		Slew2AbsAzEl:=CmdResponseType.CommandActivated;	
	ELSE 
		Slew2AbsAzEl:=CmdResponseType.ParameterOutOfRange;
	END_IF			   
END_IF
r_write_position_az_out:=Pos_Az; // Writeing setpoint positions to Cyclic out put to get P.Set outputs
r_write_position_el_out:=Pos_El;
CommandArbiter.Status.LastCmdResponse:=Slew2AbsAzEl;
END_METHOD

METHOD Slew2AbsSingleAx : UINT
VAR_INPUT
	SessionID: UINT;
	Axis: Uint;
	Position:LREAL;
	Speed:LREAL;
END_VAR

VAR
END_VAR
CASE CommandArbiter.Status.DscCmdAuthority OF                    // Check that correct user is issueing a command
	LMC: IF SessionID= CommandArbiter.Lmc_ID THEN
			Slew2AbsSingleAx:= CmdResponseType.CommandActivated;
     	 END_IF
			
	EGUI: IF SessionID= CommandArbiter.Egui_ID THEN
			Slew2AbsSingleAx:= CmdResponseType.CommandActivated;
    	  END_IF		
ELSE 
     Slew2AbsSingleAx:= CmdResponseType.NoCmdAuth;
     Command_Arbiter_error:=1;	
END_CASE

IF Slew2AbsSingleAx = CmdResponseType.CommandActivated THEN // Dish State to see if move is possible
	Command_Arbiter_error:=0;
	//IF  Management.ErrorStatus.errGeneral=0 AND Management.WarningStatus.waMngmnt =0 THEN   If the Dish has errors that prevent movement then it will not be in a state where it can be moved. 
		CASE Management.Status.DscState OF 
			 DscStateType.Locked:        Slew2AbsSingleAx:=CmdResponseType.DishLocked;
			 DscStateType.Locked_Stowed: Slew2AbsSingleAx:=CmdResponseType.DishLocked;
			 DscStateType.Standstill:    Slew2AbsSingleAx:=CmdResponseType.CommandActivated;
		     DscStateType.Standby:       Slew2AbsSingleAx:=CmdResponseType.CommandActivated;
			 DscStateType.Stowed:	IF Axis=2 THEN 
				Slew2AbsSingleAx:= CmdResponseType.CommandActivated;
			ELSE
		 	Slew2AbsSingleAx:=CmdResponseType.Stowed;
			END_IF
  
		ELSE
		     Slew2AbsSingleAx:=CmdResponseType.CommandRejected;
		     Command_Arbiter_error:=1;
		END_CASE								
	//ELSE
	//	Slew2AbsAx:=CmdResponseType.CommandAborted;
	//	Command_Arbiter_error:=1;
	//END_IF
END_IF
	
IF Slew2AbsSingleAx = CmdResponseType.CommandActivated THEN  // Move selected axis
	b_goto_rel:=FALSE;
	CASE Axis OF 
		AxisSelectType.Az:	
            IF (Position <= gc_r_pos_max_Az) AND (Position>= gc_r_pos_min_Az) AND (Speed <= gc_r_vel_max_Az*6) THEN
           		b_activate_Az:=1;
			    r_goto_Az := LREAL_TO_REAL(Position);
				 IF Speed > r_vel_max_Az THEN    // For power management
					 r_goto_v_Az:= r_vel_max_Az;
				 ELSE
				 	 r_goto_v_Az:= LREAL_TO_REAL(Speed/6); 
				 END_IF
				b_stop_Az:= FALSE;
				b_start_goto_Az:= TRUE;
				Slew2AbsSingleAx:=CmdResponseType.CommandActivated;
				r_write_position_az_out:=Position; // Writeing setpoint positions to Cyclic out put to get P.Set outputs
			ELSE 
				Slew2AbsSingleAx:=CmdResponseType.ParameterOutOfRange;
			END_IF			   
		AxisSelectType.El:
 			IF (Position <= gc_r_pos_max_El) AND (Position>= gc_r_pos_min_El) AND (Speed <= gc_r_vel_max_El*6
) THEN
            	b_activate_el:=1;
				r_goto_El := LREAL_TO_REAL(Position);
				
				 IF Speed > r_vel_max_El THEN    // For power management
					 r_goto_v_El:= r_vel_max_El;
				 ELSE
				 	 r_goto_v_El:= LREAL_TO_REAL(Speed/6); 
				 END_IF
				
				b_stop_El:= FALSE;
				b_start_goto_El:= TRUE;
				Slew2AbsSingleAx:=CmdResponseType.CommandActivated;
				r_write_position_el_out:=Position; // Writeing setpoint positions to Cyclic out put to get P.Set outputs
			ELSE 
				Slew2AbsSingleAx:=CmdResponseType.ParameterOutOfRange;
			END_IF 
					    
		AxisSelectType.FI: 
			IF (Position <= gc_r_pos_max_Fi) AND (Position >= gc_r_pos_min_Fi) AND (Speed<= gc_r_vel_max_Fi*6) THEN
                 b_activate_Fi:=1;
				 r_goto_Fi := LREAL_TO_REAL(Position);
				 IF Speed > r_vel_max_Fi THEN 
					 r_goto_v_Fi:= r_vel_max_Fi;
				 ELSE
				 	 r_goto_v_Fi:= LREAL_TO_REAL(Speed/6); 
				 END_IF
				 b_stop_Fi:= FALSE;
				 b_start_goto_Fi:= TRUE;
				 Slew2AbsSingleAx:=CmdResponseType.CommandActivated;
				 r_write_position_fi_out:=Position; // Writeing setpoint positions to Cyclic out put to get P.Set outputs
		    ELSE 
				 Slew2AbsSingleAx:=CmdResponseType.ParameterOutOfRange;
			END_IF              
 			     									
	ELSE
		Slew2AbsSingleAx:=CmdResponseType.ParameterOutOfRange;
	END_CASE
END_IF

CommandArbiter.Status.LastCmdResponse:=Slew2AbsSingleAx;
END_METHOD

METHOD Slew2RelAzEl : UINT
VAR_INPUT
	SessionID:UINT;
	Pos_Az:LREAL;
	Pos_El:LREAL;
	Speed_Az:LREAL;
	Speed_El:LREAL;
	
END_VAR
CASE CommandArbiter.Status.DscCmdAuthority OF                    // Check that correct user is issueing a command
	LMC: IF SessionID= CommandArbiter.Lmc_ID THEN
			Slew2RelAzEl:= CmdResponseType.CommandActivated;
     	 END_IF
			
	EGUI: IF SessionID= CommandArbiter.Egui_ID THEN
			Slew2RelAzEl:= CmdResponseType.CommandActivated;
    	  END_IF		
ELSE 
     Slew2RelAzEl:= CmdResponseType.NoCmdAuth;
     Command_Arbiter_error:=1;	
END_CASE

IF Slew2RelAzEl = CmdResponseType.CommandActivated THEN // Dish State to see if move is possible
	Command_Arbiter_error:=0;
	//IF  Management.ErrorStatus.errGeneral=0 AND Management.WarningStatus.waMngmnt =0 THEN  (*The Dish in the standby state*)
		CASE Management.Status.DscState OF 
			 DscStateType.Locked:        Slew2RelAzEl:=CmdResponseType.DishLocked;
			 DscStateType.Locked_Stowed: Slew2RelAzEl:=CmdResponseType.DishLocked;
			 DscStateType.Standstill:    Slew2RelAzEl:=CmdResponseType.CommandActivated;
		     DscStateType.Standby:       Slew2RelAzEl:=CmdResponseType.CommandActivated;
			 DscStateType.Stowed:	     Slew2RelAzEl:=CmdResponseType.Stowed;
		ELSE
		     Slew2RelAzEl:=CmdResponseType.CommandRejected;
		     Command_Arbiter_error:=1;
		END_CASE								
	(*ELSE
		Slew2RelAzEl:=CmdResponseType.CommandAborted;
		Command_Arbiter_error:=1;
	END_IF *)
END_IF
	
IF Slew2RelAzEl = CmdResponseType.CommandActivated THEN  // Move selected axis
	IF (((Pos_Az + r_pos_az_v) <= gc_r_pos_max_Az) AND ((Pos_Az + r_pos_az_v )>= gc_r_pos_min_Az) AND ( Speed_Az <= gc_r_vel_max_Az*6)) AND (((Pos_El + r_pos_el_v) <= gc_r_pos_max_El) AND ((Pos_El + r_pos_el_v )>= gc_r_pos_min_El) AND ( Speed_El <= gc_r_vel_max_El*6)) THEN
    	b_activate_Az:=1;
		r_goto_Az := LREAL_TO_REAL(Pos_Az);
		b_goto_rel:=TRUE;
		r_goto_v_Az:= LREAL_TO_REAL(Speed_Az/6); 
		b_stop_Az:= FALSE;
		b_start_goto_Az:= TRUE;
		b_activate_el:=1;
		r_goto_El := LREAL_TO_REAL(Pos_El);
		r_goto_v_El:= LREAL_TO_REAL(Speed_El/6); 
		b_stop_El:= FALSE;
		b_start_goto_El:= TRUE;
		Slew2RelAzEl:=CmdResponseType.CommandActivated;	
	ELSE 
		Slew2RelAzEl:=CmdResponseType.ParameterOutOfRange;
	END_IF			   
	
END_IF

CommandArbiter.Status.LastCmdResponse:=Slew2RelAzEl;
END_METHOD

METHOD Slew2RelSingleAx : UINT
VAR_INPUT
	SessionID:UINT;
	Axis: UINT;
	Position:LREAL;
	Speed:LREAL;
END_VAR
CASE CommandArbiter.Status.DscCmdAuthority OF                    // Check that correct user is issueing a command
	LMC: IF SessionID= CommandArbiter.Lmc_ID THEN
			Slew2RelSingleAx:= CmdResponseType.CommandActivated;
     	 END_IF
			
	EGUI: IF SessionID= CommandArbiter.Egui_ID THEN
			Slew2RelSingleAx:= CmdResponseType.CommandActivated;
    	  END_IF		
ELSE 
     Slew2RelSingleAx:= CmdResponseType.NoCmdAuth;
     Command_Arbiter_error:=1;	
END_CASE

IF Slew2RelSingleAx = CmdResponseType.CommandActivated THEN // Dish State to see if move is possible
	Command_Arbiter_error:=0;
	//IF  Management.ErrorStatus.errGeneral=0 AND Management.WarningStatus.waMngmnt =0 THEN  (*The Dish in the standby state*)
		CASE Management.Status.DscState OF 
			 DscStateType.Locked:        Slew2RelSingleAx:=CmdResponseType.DishLocked;
			 DscStateType.Locked_Stowed: Slew2RelSingleAx:=CmdResponseType.DishLocked;
			 DscStateType.Standstill:    Slew2RelSingleAx:=CmdResponseType.CommandActivated;
		     DscStateType.Standby:       Slew2RelSingleAx:=CmdResponseType.CommandActivated;
			 DscStateType.Stowed:	     
								 IF Axis=2 THEN 
									Slew2RelSingleAx:= CmdResponseType.CommandActivated;
								 ELSE
		 							Slew2RelSingleAx:=CmdResponseType.Stowed;
								 END_IF
			
		ELSE
		     Slew2RelSingleAx:=CmdResponseType.CommandRejected;
		     Command_Arbiter_error:=1;
		END_CASE								
(*	ELSE
		Slew2RelAx:=CmdResponseType.CommandAborted;
		Command_Arbiter_error:=1;
	END_IF*)
END_IF
	
IF Slew2RelSingleAx = CmdResponseType.CommandActivated THEN  // Move selected axis
	CASE Axis OF 
		AxisSelectType.Az:	
            IF ((Position + r_pos_az_v) <= gc_r_pos_max_Az) AND ((Position + r_pos_az_v )>= gc_r_pos_min_Az) AND ( Speed <= gc_r_vel_max_Az*6) THEN
           		b_activate_Az:=1;
			    r_goto_Az := LREAL_TO_REAL(Position);
				r_goto_v_Az:= LREAL_TO_REAL(Speed/6); 
				b_stop_Az:= FALSE;
				b_start_goto_Az:= TRUE;
				b_goto_rel:=TRUE;
				Slew2RelSingleAx:=CmdResponseType.CommandActivated;
			ELSE 
				Slew2RelSingleAx:=CmdResponseType.ParameterOutOfRange;
			END_IF			   
		AxisSelectType.El:
 			IF ((Position + r_pos_el_v) <= gc_r_pos_max_El) AND ((Position + r_pos_el_v )>= gc_r_pos_min_El) AND ( Speed <= gc_r_vel_max_El*6) THEN
            	b_activate_el:=1;
				r_goto_El := LREAL_TO_REAL(Position);
				r_goto_v_El:= LREAL_TO_REAL(Speed/6); 
				b_stop_El:= FALSE;
				b_start_goto_El:= TRUE;
				b_goto_rel:=TRUE;
				Slew2RelSingleAx:=CmdResponseType.CommandActivated;
			ELSE 
				Slew2RelSingleAx:=CmdResponseType.ParameterOutOfRange;
			END_IF 
					    
		AxisSelectType.FI: 
			IF ((Position + r_pos_fi_v) <= gc_r_pos_max_Fi) AND ((Position + r_pos_fi_v )> gc_r_pos_min_Fi) AND ( Speed <= gc_r_vel_max_Fi*6) THEN
                 b_activate_Fi:=1;
				 r_goto_Fi := LREAL_TO_REAL(Position);
				 r_goto_v_Fi:= LREAL_TO_REAL(Speed/6); 
				 b_stop_Fi:= FALSE;
				 b_start_goto_Fi:= TRUE;
				 b_goto_rel:=TRUE;
				 Slew2RelSingleAx:=CmdResponseType.CommandActivated;
		    ELSE 
				 Slew2RelSingleAx:=CmdResponseType.ParameterOutOfRange;
			END_IF              
 			     									
	ELSE
		Slew2RelSingleAx:=CmdResponseType.ParameterOutOfRange;
	END_CASE
	
		
END_IF
CommandArbiter.Status.AxisSelect:=Axis;
CommandArbiter.Status.LastCmdResponse:=Slew2RelSingleAx;
END_METHOD

METHOD Stop : UINT
VAR_INPUT
	SessionID:Uint;
	Axis: UINT; 
END_VAR
VAR_OUTPUT
	
END_VAR
VAR
	
END_VAR
CASE CommandArbiter.Status.DscCmdAuthority OF                    // Check that corerct user is issueing a command
	LMC: IF SessionID= CommandArbiter.Lmc_ID THEN
			Stop:= CmdResponseType.CommandActivated;
     	 END_IF
			
	EGUI: IF SessionID= CommandArbiter.Egui_ID THEN
			Stop:= CmdResponseType.CommandActivated;
    	  END_IF		
ELSE 
     Stop:= CmdResponseType.NoCmdAuth;
     Command_Arbiter_error:=1;	
END_CASE

IF Stop = CmdResponseType.CommandActivated THEN
	Command_Arbiter_error:=0;
	CASE Management.Status.DscState OF 
		DSCStateType.StartUp:
		 	Stop := CmdResponseType.CommandRejected;
		DSCStateType.Standby:
		 	Stop := CmdResponseType.CommandRejected;
		DSCStateType.Locked:
		 	Stop := CmdResponseType.DishLocked;
		DSCStateType.Stowed:
		 	Stop :=CmdResponseType.Stowed;
		DSCStateType.Locked_Stowed:
		 	Stop := CmdResponseType.DishLocked; 
		DSCStateType.Activating :
		 	Stop := CmdResponseType.CommandRejected;
		DSCStateType.Deactivating :
		 	Stop := CmdResponseType.CommandRejected;
		DSCStateType.Standstill :
		 	Stop := CmdResponseType.CommandActivated;
		DSCStateType.Stopping :
		 	Stop := CmdResponseType.CommandActivated;
		DSCStateType.Slew :
		 	Stop := CmdResponseType.CommandActivated;
		DSCStateType.Jog :
		 	Stop := CmdResponseType.CommandActivated;
		DSCStateType.Track :
		 	Stop := CmdResponseType.CommandActivated;
	END_CASE

	IF Stop = CmdResponseType.CommandActivated THEN
		b_track_on:=0; // In case a track is runnning then stop the track
		CASE Axis OF
			AxisSelectType.Unknown:  // Stops all 
		       b_scc_stop:=1;
			    b_start_goto_Fi:=0;
			AxisSelectType.Az:
			  b_stop_Az:=1;
			  b_start_goto_Az:=0;
			AxisSelectType.El:
			 b_stop_El:=1;
			 b_start_goto_El:=0;
			AxisSelectType.Fi:
			 b_stop_Fi:=1;
			 b_start_goto_Fi:=0;
			AxisSelectType.AzEl:
			  b_scc_stop:=1;
			   b_stop_Az:=1;
			   b_stop_El:=1;
			   b_start_goto_El:=0;
			   b_start_goto_Az:=0;
		ELSE
			Stop := CmdResponseType.ParameterOutOfRange;
		END_CASE
	END_IF 
			
END_IF
CommandArbiter.Status.LastCmdResponse:= Stop;
END_METHOD

METHOD Stow : Uint
VAR_INPUT
	SessionID:UINT;
	StowAction:BOOL;
END_VAR


VAR
	Speed_El: REAL;
	Speed_Az: Real;
END_VAR
CASE CommandArbiter.Status.DscCmdAuthority OF                    // Check that correct user is issueing a command
	LMC: IF SessionID= CommandArbiter.Lmc_ID THEN
			Stow:= CmdResponseType.CommandActivated;
     	 END_IF
			
	EGUI: IF SessionID= CommandArbiter.Egui_ID THEN
			Stow:= CmdResponseType.CommandActivated;
    	  END_IF		
ELSE 
     Stow:= CmdResponseType.NoCmdAuth;
     Command_Arbiter_error:=1;	
END_CASE

IF Stow = CmdResponseType.CommandActivated THEN // Dish State to see if move is possible
	Command_Arbiter_error:=0;
	IF  Management.ErrorStatus.errGeneral=0 AND Management.WarningStatus.waMngmnt =0 THEN  (*The Dish in the standby state*)
		CASE Management.Status.DscState OF 
			 DscStateType.Locked:        Stow:=CmdResponseType.DishLocked;
			 DscStateType.Locked_Stowed: Stow:=CmdResponseType.DishLocked;
			 DscStateType.Standstill:    Stow:=CmdResponseType.CommandActivated;
		     DscStateType.Standby:       Stow:=CmdResponseType.CommandActivated;
			 DscStateType.Slew:          Stow:=CmdResponseType.CommandActivated;
			 DscStateType.Track:         Stow:=CmdResponseType.CommandActivated;
			                              //Stop Track
			 DscStateType.Stowed:	     Stow:=CmdResponseType.CommandActivated;
		ELSE
		     Stow:=CmdResponseType.CommandRejected;
		     Command_Arbiter_error:=1;
		END_CASE								
	ELSE
		Stow:=CmdResponseType.CommandRejected;
		Command_Arbiter_error:=1;
	END_IF
END_IF

IF Stow = CmdResponseType.CommandActivated THEN
	IF StowAction = TRUE THEN 
		b_activate_Az:=1;
		b_activate_el:=1;
		b_stow:=1; 
		
		IF b_UPS_stow THEN 
		   Speed_Az:= gc_UPS_Stow_Az_Speed;
	       Speed_El:=gc_UPS_Stow_El_Speed; 
		ELSE
		   Speed_Az:= gc_r_vel_max_Az;
	       Speed_El:=gc_r_vel_max_El; 
		END_IF
		
		//r_goto_Az := LREAL_TO_REAL(0-r_pos_az_v);
		r_goto_Az :=0;
		r_goto_v_Az:= LREAL_TO_REAL(Speed_Az); 
		r_goto_El := 90;
		r_goto_v_El:= LREAL_TO_REAL(Speed_El); 
		
		
        b_stop_Az:= FALSE;
		//b_start_goto_Az:= TRUE;
		b_stop_El:= FALSE;
		//b_start_goto_El:= TRUE;
		
      // Activates ladder logic A_STOW
		b_stow_pin_retract:=0;	
		
		Stow:=CmdResponseType.CommandActivated;	
	ELSIF StowAction = FALSE THEN 
		b_stow_pin_retract:=1 ;
		//b_stow:= 0;	
	END_IF
END_IF
	
r_write_position_az_out:=0; // Writeing setpoint positions to Cyclic out put to get P.Set outputs
r_write_position_el_out:=90;	

CommandArbiter.Status.LastCmdResponse:=Stow;
END_METHOD

METHOD TrackStartDM : UINT
VAR_INPUT
	SessionID:UINT;
	Interpol :UINT; // 0 = Newton 1= Spline
	StartTime : LREAL ;
	
END_VAR
CASE CommandArbiter.Status.DscCmdAuthority OF                    // Check that corerct user is issueing a command
	LMC: IF SessionID= CommandArbiter.Lmc_ID THEN
			TrackStartDM:= CmdResponseType.CommandActivated;
     	 END_IF
			
	EGUI: IF SessionID= CommandArbiter.Egui_ID THEN
			TrackStartDM:= CmdResponseType.CommandActivated;
    	  END_IF		
ELSE 
     TrackStartDM:= CmdResponseType.NoCmdAuth;
     Command_Arbiter_error:=1;	
END_CASE


IF TrackStartDM = CmdResponseType.CommandActivated THEN // Dish State to see if move is possible
	Command_Arbiter_error:=0;
	IF  Management.ErrorStatus.errGeneral=0 AND Management.WarningStatus.waMngmnt =0 THEN  (*The Dish in the standby state*)
		CASE Management.Status.DscState OF 
			 DscStateType.Locked:        TrackStartDM:=CmdResponseType.DishLocked;
			 DscStateType.Locked_Stowed: TrackStartDM:=CmdResponseType.DishLocked;
			 DscStateType.Standstill:    TrackStartDM:=CmdResponseType.CommandActivated;
		     DscStateType.Standby:       TrackStartDM:=CmdResponseType.CommandActivated;
			 DscStateType.Stowed:	     TrackStartDM:=CmdResponseType.Stowed;
		ELSE
		     TrackStartDM:=CmdResponseType.CommandRejected;
		     Command_Arbiter_error:=1;
		END_CASE								
	ELSE
		TrackStartDM:=CmdResponseType.CommandRejected;
		Command_Arbiter_error:=1;
	END_IF
END_IF


IF TrackStartDM= CmdResponseType.CommandActivated AND(StartTime> Time_cds.Status.TAIoffset) THEN
	TrackStartDM:=CmdResponseType.CommandActivated;	
	b_track_start:=1;
	lr_track_start_time:=StartTime;
ELSIF StartTime < 0 THEN  // Times can't be less than zero
	TrackStartDM:=CmdResponseType.ParameterOutOfRange;
ELSE 	
	TrackStartDM:=CmdResponseType.CommandActivated;	
	b_track_start:=1;
	lr_track_start_time:=Time_cds.Status.TAIoffset+0.1; // add 100ms to give enough time to start track. 
END_IF			   



CommandArbiter.Status.LastCmdResponse:=TrackStartDM;
END_METHOD

METHOD TrackStartPolyDM : UINT
VAR_INPUT
	SessionID: UINT;
	TrackId: UINT; 
	Order : UINT;
		
END_VAR
CASE CommandArbiter.Status.DscCmdAuthority OF                    // Check that corerct user is issueing a command
	LMC: IF SessionID= CommandArbiter.Lmc_ID THEN
			TrackStartPolyDM:= CmdResponseType.CommandActivated;
     	 END_IF
			
	EGUI: IF SessionID= CommandArbiter.Egui_ID THEN
			TrackStartPolyDM:= CmdResponseType.CommandActivated;
    	  END_IF		
ELSE 
    TrackStartPolyDM:= CmdResponseType.NoCmdAuth;
     Command_Arbiter_error:=1;	
END_CASE


TrackStartPolyDM:=CmdResponseType.NotImplemented;
CommandArbiter.Status.LastCmdResponse:=TrackStartPolyDM;
END_METHOD

END_FUNCTION_BLOCK

// IndraMotionMlc1/Application/POUs/OPCUA/OPCUA_Method/fb_Pointing
(*{attribute 'opcua.mapping.type' := ''}
{attribute 'opcua.mapping.modeluri' := 'http://skao.int/DS_ICD/'}
{attribute 'opcua.mapping.publicationdate' := '12/14/2023 00:00:00'}
{attribute 'opcua.mapping.nodeid' := 'nsu=http://skao.int/DS_ICD/;i=1014'}*)
FUNCTION_BLOCK fb_Pointing
VAR_INPUT
	Commands: fb_Pointing_Commands;
	Status: PointingStatus_Type;
	AmbTempParameters: AmbTempParam_Type;
	StaticPmParameters: ARRAY [0..7] OF StaticPmParam;
	TiltmeterParameters: TiltmeterParam;
	
	
	
END_VAR
VAR
	TE :LREAL:=0; 
	
END_VAR

END_FUNCTION_BLOCK

// IndraMotionMlc1/Application/POUs/OPCUA/OPCUA_Method/fb_Pointing_Commands
(*{attribute 'opcua.mapping.type' := ''}
{attribute 'opcua.mapping.modeluri' := 'http://skao.int/DS_ICD/'}
{attribute 'opcua.mapping.publicationdate' := '12/14/2023 00:00:00'}
{attribute 'opcua.mapping.nodeid' := 'nsu=http://skao.int/DS_ICD/;i=1014'}*)
FUNCTION_BLOCK fb_Pointing_Commands
VAR_INPUT
	
END_VAR

METHOD AmbTempCorrSetup : UINT

VAR_INPUT
	SessionID:Uint;
	filt_dt:LREAL;
	ambTempParam1:LREAL;
	ambTempParam2:LREAL;
	ambTempParam3:LREAL;
	ambTempParam4:LREAL;
	ambTempParam5:LREAL;
	ambTempParam6:LREAL;
END_VAR
VAR_OUTPUT
	
END_VAR
VAR
END_VAR
IF SessionID = CommandArbiter.Egui_ID AND CommandArbiter.Status.DscCmdAuthority= EGUI THEN
	Command_Arbiter_error:=0;
	IF filt_dt>=0 AND  filt_dt<=1000 THEN         // Only checks if filt_dt is in range
		Pointing.AmbTempParameters.filt_dt:=filt_dt;
		Pointing.AmbTempParameters.ambTempParam1:=ambTempParam1;
		Pointing.AmbTempParameters.ambTempParam2:=ambTempParam2;
		Pointing.AmbTempParameters.ambTempParam3:=ambTempParam3;
		Pointing.AmbTempParameters.ambTempParam4:=ambTempParam4;
		Pointing.AmbTempParameters.ambTempParam5:=ambTempParam5;
		Pointing.AmbTempParameters.ambTempParam6:=ambTempParam6;	
		AmbTempCorrSetup:=CmdResponseType.CommandDone;
	ELSE
		AmbTempCorrSetup:=CmdResponseType.ParameterOutOfRange;		
	END_IF
ELSE
  AmbTempCorrSetup:=CmdResponseType.NoCmdAuth;
Command_Arbiter_error:=1;	
END_IF

CommandArbiter.Status.LastCmdResponse:= AmbTempCorrSetup;
END_METHOD

METHOD PmCorrOnOff : UINT

VAR_INPUT
	SessionID:UINT;
	StaticOn:BOOL;
	TiltOn:UINT;
	AmbTOn:BOOL;
	Band:UINT;
	
END_VAR
VAR_OUTPUT
	
END_VAR
VAR
END_VAR
CASE CommandArbiter.Status.DscCmdAuthority OF                    // Check that corerct user is issueing a command
	LMC: IF SessionID= CommandArbiter.Lmc_ID THEN
			PmCorrOnOff:= CmdResponseType.CommandActivated;
         END_IF
			
	EGUI: IF SessionID= CommandArbiter.Egui_ID THEN
			PmCorrOnOff:= CmdResponseType.CommandActivated;
     	  END_IF		
ELSE 
     PmCorrOnOff:= CmdResponseType.NoCmdAuth;
     Command_Arbiter_error:=1;	
END_CASE

IF PmCorrOnOff = CmdResponseType.CommandActivated THEN 
	IF  Band <8 AND Band >= 0 THEN 
		Command_Arbiter_error:=0;
		Pointing.Status.BandForCorr:=Band;
		PmCorrOnOff:=CmdResponseType.CommandDone;
		IF StaticOn THEN
	    	Pointing.Status.StaticCorrActive:=TRUE;
		ELSE
			Pointing.Status.StaticCorrActive:=FALSE;		
		END_IF
		
		IF AmbTOn THEN
			Pointing.Status.AmbTempCorrActive:=TRUE;
		ELSE
			Pointing.Status.AmbTempCorrActive:=FALSE;	
		END_IF
	
		CASE TiltOn OF
        	0: Pointing.Status.TiltCorrActive:=0;
			   Pointing.Status.TiltOne_On:=0;
			   Pointing.Status.TiltTwo_On:=0;
						
        	1: Pointing.Status.TiltCorrActive:=1;
		   	   Pointing.Status.TiltOne_On:=1;
			   Pointing.Status.TiltTwo_On:=0;
			   
			2: Pointing.Status.TiltCorrActive:=1;
		   	   Pointing.Status.TiltOne_On:=0;
			   Pointing.Status.TiltTwo_On:=1;
   	 	ELSE
			PmCorrOnOff:=CmdResponseType.ParameterOutOfRange;
		END_CASE
	   
	ELSE 
		PmCorrOnOff:=CmdResponseType.ParameterOutOfRange;
	END_IF
END_IF
CommandArbiter.Status.LastTiltOn:=TiltOn;
CommandArbiter.Status.LastCmdResponse:= PmCorrOnOff;
END_METHOD

METHOD StaticPmSetup : UINT
VAR_INPUT
	SessionID:UINT;
	Band:UINT;
	IA:LREAL;
	CA:LREAL;
	NPAE:LREAL;
	AN:LREAL;
	AN0:LREAL;
	AW:LREAL;
	AW0:LREAL;
	ACEC:LREAL;
	ACES:LREAL;
	ABA:LREAL;
	ABphi:LREAL;
	IE:LREAL;
	ECEC: LREAL;
	ECES: LREAL;
	HECE4: LREAL;
	HESE4:LREAL;
	HECE8:LREAL;
	HESE8:LREAL;

END_VAR
VAR_OUTPUT
	
END_VAR
VAR
END_VAR
CASE CommandArbiter.Status.DscCmdAuthority OF                    // Check that corerct user is issueing a command
	LMC: IF SessionID= CommandArbiter.Lmc_ID THEN
			StaticPmSetup:= CmdResponseType.CommandActivated;
         END_IF
			
	EGUI: IF SessionID= CommandArbiter.Egui_ID THEN
			StaticPmSetup:= CmdResponseType.CommandActivated;
     	  END_IF		
ELSE 
     StaticPmSetup:= CmdResponseType.NoCmdAuth;
     Command_Arbiter_error:=1;	
END_CASE



IF StaticPmSetup = CmdResponseType.CommandActivated  THEN
	Command_Arbiter_error:=0;
	IF Band >=0 AND Band <8 THEN
		Pointing.StaticPmParameters[Band].IA:=IA;
		Pointing.StaticPmParameters[Band].CA:=CA;
		Pointing.StaticPmParameters[Band].NPAE:=NPAE;
		Pointing.StaticPmParameters[Band].AN:=AN;
		Pointing.StaticPmParameters[Band].AN0:=AN0;
		Pointing.StaticPmParameters[Band].AW:=AW;
		Pointing.StaticPmParameters[Band].AW0:=AW0;
		Pointing.StaticPmParameters[Band].ACEC:=ACEC;
		Pointing.StaticPmParameters[Band].ACES:=ACES;
		Pointing.StaticPmParameters[Band].ABA:=ABA;
		Pointing.StaticPmParameters[Band].ABphi:=ABphi;
		Pointing.StaticPmParameters[Band].IE:=IE;
		Pointing.StaticPmParameters[Band].ECEC:=ECEC;
		Pointing.StaticPmParameters[Band].ECES:=ECES;
		Pointing.StaticPmParameters[Band].HECE4:=HECE4;
		Pointing.StaticPmParameters[Band].HESE4:=HESE4;
		Pointing.StaticPmParameters[Band].HECE8:=HECE8;
		Pointing.StaticPmParameters[Band].HESE8:=HESE8;
		StaticPmSetup:=CmdResponseType.CommandDone;
	ELSE
   		StaticPmSetup:=CmdResponseType.ParameterOutOfRange;	
	END_IF
ELSE
   StaticPmSetup:=CmdResponseType.NoCmdAuth;	
   Command_Arbiter_error:=1;
END_IF
CommandArbiter.Status.LastCmdResponse:=StaticPmSetup;
END_METHOD

METHOD TiltCalSetup : UINT
VAR_INPUT
	SessionID:Uint;
	TiltmeterPos:UINT;
	Tiltmeter_serial_no:STRING;
	tilt_temp_scale:LREAL;
	x_filt_dt:LREAL;
	x_off:LREAL;
	x_offTC:LREAL;
	x_scale:LREAL;
	x_scaleTC:LREAL;
	x_zero:LREAL;
	x_zeroTC:LREAL;
	y_filt_dt:LREAL;
	y_off:LREAL;
	y_offTC:LREAL;
	y_scale:LREAL;
	y_scaleTC:LREAL;
	y_zero:LREAL;
	y_zeroTC:LREAL;
	
	
END_VAR
VAR_OUTPUT
	
END_VAR
VAR
END_VAR
IF SessionID = CommandArbiter.Egui_ID AND CommandArbiter.Status.DscCmdAuthority = EGUI THEN
	Command_Arbiter_error:=0;
	IF TiltmeterPos=1  THEN
		Pointing.TiltmeterParameters.One.Tiltmeter_serial_no:=Tiltmeter_serial_no;
		Pointing.TiltmeterParameters.One.Tilt_temp_scale:=Tilt_temp_scale;
		Pointing.TiltmeterParameters.One.x_scale:=x_scale;
		Pointing.TiltmeterParameters.One.x_scaleTC:=x_scaleTC;
		Pointing.TiltmeterParameters.One.x_zero:=x_zero;
		Pointing.TiltmeterParameters.One.x_zeroTC:=x_zeroTC;
		Pointing.TiltmeterParameters.One.x_off:=x_off;
		Pointing.TiltmeterParameters.One.x_offTC:=x_offTC;
		Pointing.TiltmeterParameters.One.x_filt_dt:=x_filt_dt;
		Pointing.TiltmeterParameters.One.y_scale:=y_scale;
		Pointing.TiltmeterParameters.One.y_scaleTC:=y_scaleTC;
		Pointing.TiltmeterParameters.One.y_zero:=y_zero;
		Pointing.TiltmeterParameters.One.y_zeroTC:=y_zeroTC;
		Pointing.TiltmeterParameters.One.y_off:=y_off;
		Pointing.TiltmeterParameters.One.y_offTC:=y_offTC;
		Pointing.TiltmeterParameters.One.y_filt_dt:=y_filt_dt;
		TiltCalSetup:=CmdResponseType.CommandDone;
	ELSIF TiltmeterPos=2  THEN
		Pointing.TiltmeterParameters.Two.Tiltmeter_serial_no:=Tiltmeter_serial_no;
		Pointing.TiltmeterParameters.Two.Tilt_temp_scale:=Tilt_temp_scale;
		Pointing.TiltmeterParameters.Two.x_scale:=x_scale;
		Pointing.TiltmeterParameters.Two.x_scaleTC:=x_scaleTC;
		Pointing.TiltmeterParameters.Two.x_zero:=x_zero;
		Pointing.TiltmeterParameters.Two.x_zeroTC:=x_zeroTC;
		Pointing.TiltmeterParameters.Two.x_off:=x_off;
		Pointing.TiltmeterParameters.Two.x_offTC:=x_offTC;
		Pointing.TiltmeterParameters.Two.x_filt_dt:=x_filt_dt;
		Pointing.TiltmeterParameters.Two.y_scale:=y_scale;
		Pointing.TiltmeterParameters.Two.y_scaleTC:=y_scaleTC;
		Pointing.TiltmeterParameters.Two.y_zero:=y_zero;
		Pointing.TiltmeterParameters.Two.y_zeroTC:=y_zeroTC;
		Pointing.TiltmeterParameters.Two.y_off:=y_off;
		Pointing.TiltmeterParameters.Two.y_offTC:=y_offTC;
		Pointing.TiltmeterParameters.Two.y_filt_dt:=y_filt_dt;
		TiltCalSetup:=CmdResponseType.CommandDone;	
	ELSE
		TiltCalSetup:=CmdResponseType.ParameterOutOfRange;		
	END_IF
ELSE
   TiltCalSetup:=CmdResponseType.NoCmdAuth;	
   Command_Arbiter_error:=1;
END_IF

CommandArbiter.Status.LastCmdResponse:=TiltCalSetup;
END_METHOD

END_FUNCTION_BLOCK

// IndraMotionMlc1/Application/POUs/OPCUA/OPCUA_Method/fb_Safety
(*{attribute 'opcua.mapping.type' := ''}
{attribute 'opcua.mapping.modeluri' := 'http://skao.int/DS_ICD/'}
{attribute 'opcua.mapping.publicationdate' := '12/14/2023 00:00:00'}
{attribute 'opcua.mapping.nodeid' := 'nsu=http://skao.int/DS_ICD/;i=1012'}*)
FUNCTION_BLOCK fb_Safety
VAR_INPUT	
	Commands: fb_Safety_Commands;
	Status: SafetyStatus_Type;
	
END_VAR

END_FUNCTION_BLOCK

// IndraMotionMlc1/Application/POUs/OPCUA/OPCUA_Method/fb_Safety_Commands
(*{attribute 'opcua.mapping.type' := ''}
{attribute 'opcua.mapping.modeluri' := 'http://skao.int/DS_ICD/'}
{attribute 'opcua.mapping.publicationdate' := '12/14/2023 00:00:00'}
{attribute 'opcua.mapping.nodeid' := 'nsu=http://skao.int/DS_ICD/;i=1012'}*)
FUNCTION_BLOCK fb_Safety_Commands
VAR_INPUT	
	
	
END_VAR

METHOD InterlockAck :UINT
VAR_INPUT
	SessionID:UINT;	
END_VAR
VAR_OUTPUT
	
END_VAR
VAR
	b_clear_interlock:BOOL;
	
END_VAR
CASE CommandArbiter.Status.DscCmdAuthority OF                    // Check that corerct user is issueing a command
	LMC: IF SessionID = CommandArbiter.Lmc_ID THEN
			InterlockAck:= CmdResponseType.CommandActivated;
         END_IF
			
	EGUI: IF SessionID = CommandArbiter.Egui_ID THEN
		     InterlockAck:= CmdResponseType.CommandActivated;
          END_IF		
ELSE 
     InterlockAck:= CmdResponseType.NoCmdAuth;
     Command_Arbiter_error:=1;	
END_CASE

IF InterlockAck = CmdResponseType.CommandActivated THEN     // Check if the Command can be used in the current dish state
	CASE Management.Status.DscState OF 
		DSCStateType.Locked:
		 	InterlockAck := CmdResponseType.CommandActivated;
		DSCStateType.Locked_Stowed:
		 	InterlockAck := CmdResponseType.CommandActivated;
	ELSE
		InterlockAck := CmdResponseType.CommandFailed;
		Command_Arbiter_error:=1;	
	END_CASE
END_IF

IF InterlockAck = CmdResponseType.CommandActivated THEN   // Clear the interlocks
	Command_Arbiter_error:=0;
  IF  Safety.Status.InterlockClearable THEN
	//b_clear_interlock:=1;
	b_Estop_active:=0;
	b_interlock_active_Az:=0;
	b_interlock_active_El:=0;
	b_interlock_active_Fi:=0;
	Safety.Status.InterlockClearable:=0;
	InterlockAck:=CmdResponseType.CommandDone;		
  ELSE 
	InterlockAck:=CmdResponseType.CommandRejected;
	b_clear_interlock:=0;
  END_IF
END_IF

CommandArbiter.Status.LastCmdResponse:= InterlockAck;
END_METHOD

METHOD MoveStowPin :UINT
VAR_INPUT	
	SessionID: UINT;
	StowPinDeploy:BOOL;
END_VAR
	
VAR_OUTPUT
	
END_VAR
VAR
	Users:STRING;
END_VAR
CASE CommandArbiter.Status.DscCmdAuthority OF                    // Check that corerct user is issueing a command
		
	EGUI: IF SessionID = CommandArbiter.Egui_ID THEN
		     MoveStowPin:= CmdResponseType.CommandActivated;
          ELSE 
			 MoveStowPin:= CmdResponseType.NoCmdAuth;
		  END_IF		
ELSE 
     MoveStowPin:= CmdResponseType.NoCmdAuth;
     Command_Arbiter_error:=1;	
END_CASE

IF MoveStowPin = CmdResponseType.CommandActivated THEN     // Check if the Command can be used in the current dish state
	CASE Management.Status.DscState OF 
		DscStateType.StartUp:
		    MoveStowPin := CmdResponseType.CommandActivated;
		DscStateType.Standstill:
		    MoveStowPin := CmdResponseType.CommandActivated;
		DscStateType.Standby :
			MoveStowPin := CmdResponseType.CommandActivated;
		DSCStateType.Locked:
		 	MoveStowPin := CmdResponseType.DishLocked;
		DSCStateType.Locked_Stowed:
		 	MoveStowPin := CmdResponseType.DishLocked;
		DSCStateType.Stowed	:
		    MoveStowPin := CmdResponseType.CommandActivated;
	ELSE
		MoveStowPin := CmdResponseType.CommandFailed;
		Command_Arbiter_error:=1;	
	END_CASE

END_IF

IF MoveStowPin = CmdResponseType.CommandActivated AND b_stow_lock_allow THEN  // Check that Azimuth is in the correct position 
	Command_Arbiter_error:=0;
			IF StowPinDeploy= TRUE THEN
				IF b_stow_pin_limit_lock  THEN
					MoveStowPin:=CmdResponseType.Stowed;
				ELSE
					b_manual_stow:=1;
					MoveStowPin:=CmdResponseType.CommandActivated;
				END_IF		
			END_IF
	
ELSIF MoveStowPin = CmdResponseType.CommandActivated AND StowPinDeploy= FALSE THEN //Need to be able to retract Stow pin even if Encoders are in incorrect position 
	IF b_stow_pin_limit_unlock  THEN
		MoveStowPin:=CmdResponseType.CommandDone;
	ELSE
		b_manual_stow:=0;
		b_stow_pin_retract:=1;
		MoveStowPin:=CmdResponseType.CommandActivated;
	END_IF		
ELSE 
    MoveStowPin:=CmdResponseType.CommandFailed;			
END_IF		
CommandArbiter.Status.LastCmdResponse:=MoveStowPin;
END_METHOD

END_FUNCTION_BLOCK

// IndraMotionMlc1/Application/POUs/OPCUA/OPCUA_Method/fb_Time_cds
(*{attribute 'opcua.mapping.type' := ''}
{attribute 'opcua.mapping.modeluri' := 'http://skao.int/DS_ICD/'}
{attribute 'opcua.mapping.publicationdate' := '12/14/2023 00:00:00'}
{attribute 'opcua.mapping.nodeid' := 'nsu=http://skao.int/DS_ICD/;i=1023'}*)
FUNCTION_BLOCK fb_Time_cds
VAR_INPUT
	Commands: fb_Time_Commands;
	Status : Time_cdsStatus_Type;
	
END_VAR

END_FUNCTION_BLOCK

// IndraMotionMlc1/Application/POUs/OPCUA/OPCUA_Method/fb_Time_Commands
(*{attribute 'opcua.mapping.type' := ''}
{attribute 'opcua.mapping.modeluri' := 'http://skao.int/DS_ICD/'}
{attribute 'opcua.mapping.publicationdate' := '12/14/2023 00:00:00'}
{attribute 'opcua.mapping.nodeid' := 'nsu=http://skao.int/DS_ICD/;i=1023'}*)
FUNCTION_BLOCK fb_Time_Commands
VAR_INPUT
	
END_VAR

METHOD SetTimeSource : UINT
VAR_INPUT
	SessionID:  UINT;
	DscTimeSyncSource:UINT;
	TimeSourceAddrNTP:STRING;
END_VAR
VAR_OUTPUT
	
END_VAR
IF SessionID = CommandArbiter.Egui_ID AND CommandArbiter.Status.DscCmdAuthority = EGUI THEN
	Command_Arbiter_error:=0;
	CASE DscTimeSyncSource OF 
		DscTimeSyncSourceType.DSC:
			Time_cds.Status.DscTimeSyncSource:= DscTimeSyncSourceType.DSC;
			Source_Timesync:=2;
			SetTimeSource:=CmdResponseType.CommandActivated;
		DscTimeSyncSourceType.NTP:
		    Time_cds.Status.DscTimeSyncSource:= DscTimeSyncSourceType.NTP;
			Source_Timesync:=1;
			IP_Adress_NTP:=TimeSourceAddrNTP;
			SetTimeSource:=CmdResponseType.CommandActivated;
			b_ntp_update_start:=TRUE;
			
		DscTimeSyncSourceType.PTP:
			Time_cds.Status.DscTimeSyncSource:= DscTimeSyncSourceType.PTP;
			Source_Timesync:=0;
			IP_Adress_PTP:=TimeSourceAddrNTP;
			SetTimeSource:=CmdResponseType.CommandActivated;
     ELSE
		 SetTimeSource:=CmdResponseType.ParameterOutOfRange;
	END_CASE
ELSE
   SetTimeSource:=CmdResponseType.NoCmdAuth;
   Command_Arbiter_error:=1;	
END_IF

CommandArbiter.Status.LastCmdResponse:= SetTimeSource;
END_METHOD

END_FUNCTION_BLOCK

// IndraMotionMlc1/Application/POUs/OPCUA/OPCUA_Method/fb_Tracking
(*{attribute 'opcua.mapping.type' := ''}
{attribute 'opcua.mapping.modeluri' := 'http://skao.int/DS_ICD/'}
{attribute 'opcua.mapping.publicationdate' := '12/14/2023 00:00:00'}
{attribute 'opcua.mapping.nodeid' := 'nsu=http://skao.int/DS_ICD/;i=1036'}*)
FUNCTION_BLOCK fb_Tracking
VAR_INPUT
	Commands: fb_Tracking_Commands; 
	Status : TrackingStatus_Type;
	PolyStatus: PolyStatus_type;
	TableStatus: TableStatus_type;
END_VAR

END_FUNCTION_BLOCK

// IndraMotionMlc1/Application/POUs/OPCUA/OPCUA_Method/fb_Tracking_Commands
(*{attribute 'opcua.mapping.type' := ''}
{attribute 'opcua.mapping.modeluri' := 'http://skao.int/DS_ICD/'}
{attribute 'opcua.mapping.publicationdate' := '12/14/2023 00:00:00'}
{attribute 'opcua.mapping.nodeid' := 'nsu=http://skao.int/DS_ICD/;i=1036'}*)
FUNCTION_BLOCK fb_Tracking_Commands
VAR

END_VAR

METHOD TrackLoadStaticOff : Uint
VAR_INPUT
	SessionID:UINT;
	Off_Xel : LREAL;
	Off_El: LREAL;
	
END_VAR
CASE CommandArbiter.Status.DscCmdAuthority OF                    // Check that corerct user is issueing a command
	LMC: IF SessionID= CommandArbiter.Lmc_ID THEN
			TrackLoadStaticOff:= CmdResponseType.CommandActivated;
     	 END_IF
			
	EGUI: IF SessionID= CommandArbiter.Egui_ID THEN
			TrackLoadStaticOff:= CmdResponseType.CommandActivated;
    	  END_IF		
ELSE 
     TrackLoadStaticOff:= CmdResponseType.NoCmdAuth;
     Command_Arbiter_error:=1;	
END_CASE

IF TrackLoadStaticOff = CmdResponseType.CommandActivated THEN 
	IF ABS(Off_El)<= gc_r_El_off_limit AND ABS(Off_Xel)<= gc_r_Xel_off_limit THEN 
	tracking.Status.act_statOffset_value_El:=Off_El;
	tracking.Status.act_statOffset_value_Xel:=Off_Xel;
	ELSE 
		TrackLoadStaticOff:= CmdResponseType.ParameterOutOfRange;
	END_IF
END_IF

CommandArbiter.Status.LastCmdResponse:= TrackLoadStaticOff;
END_METHOD

METHOD TrackLoadTable : UINT
VAR_INPUT
	SessionID:UINT;
	LoadMode :UINT;
	SequenceLength :UINT;
    TaiOffset: ARRAY [1..1000] OF LREAL;
	Azimuth: ARRAY [1..1000] OF LREAL;
	Elevation: ARRAY [1..1000] OF LREAL;
END_VAR

VAR
 i: UINT:=1 ;
 index: UINT:=1 ;
 ValidStart: UINT:=0 ;
END_VAR

CASE CommandArbiter.Status.DscCmdAuthority OF                    // Check that corerct user is issueing a command
	LMC: IF SessionID= CommandArbiter.Lmc_ID THEN
			TrackLoadTable:= CmdResponseType.CommandActivated;
     	 END_IF
			
	EGUI: IF SessionID= CommandArbiter.Egui_ID THEN
			TrackLoadTable:= CmdResponseType.CommandActivated;
    	  END_IF		
ELSE 
     TrackLoadTable:= CmdResponseType.NoCmdAuth;
     Command_Arbiter_error:=1;	
END_CASE

IF TrackLoadTable = CmdResponseType.CommandActivated THEN 
  	IF LoadMode=0 AND(10000-i_num_stack_left) < Sequencelength THEN // Check that there is enough space in the stack.
		TrackLoadTable:= CmdResponseType.CommandFailed;
		
	ELSIF LoadMode=0 AND TaiOffset[SequenceLength] < track_table[i_End].TAIoffset THEN // Check if any point in the loaded table is at the end of the table
		TrackLoadTable:= CmdResponseType.ParameterOutOfRange;
		
	ELSE 
		FOR i:= 1 TO (SequenceLength-1) BY 1 DO    // Check that the time is monotonic 
			IF TaiOffset[i]> (TaiOffset[i+1]) THEN   
				TrackLoadTable:= CmdResponseType.NoOfParametersError;
			END_IF
		END_FOR

		FOR i:= 1 TO SequenceLength BY 1 DO  // Check that the positions are within limits
			IF ((Azimuth[i] > gc_r_pos_max_Az) OR (Azimuth[i] < gc_r_pos_min_Az)) OR ((Elevation[i] > (gc_r_pos_max_El-4)) OR (Elevation[i] < gc_r_pos_min_El)) THEN 
				TrackLoadTable:= CmdResponseType.ParameterOutOfRange;
			END_IF
		END_FOR
				
		FOR i:=(SequenceLength-1) TO 1 BY -1 DO    // Check for the time in the Sequence when the future time starts
			IF Time_cds.Status.TAIoffset < (TaiOffset[i+1]+0.1) THEN   
				ValidStart:=i;
			END_IF
		END_FOR
		IF ValidStart < 1 THEN    // Check that table has points in the future 
			TrackLoadTable:= CmdResponseType.ParameterOutOfRange;
		END_IF
	END_IF
END_IF

IF TrackLoadTable = CmdResponseType.CommandActivated THEN 
	CASE LoadMode OF
		  
		0: FOR index:= ValidStart TO SequenceLength BY 1 DO  //Append 
			 IF track_table[i_End].TAIoffset<>0 THEN 
				i_End:=F_I_number(i_End+1);
			 END_IF
			 track_table[i_End].TAIoffset:=TaiOffset[index];
			 track_table[i_End].Azimuth:= Azimuth[index];
			 track_table[i_End].Elevation:= Elevation[index];
			 
		   END_FOR  
           CommandArbiter.Status.LastLoadMode:= LoadMode; 
           
		   
		1:  i_End:= i_Start+1;  // Set the end of the table to the Start to over write the points. 
		                        // Consider adding a blend between the different tables. 
			FOR index:= ValidStart TO SequenceLength BY 1 DO  //New 
			  IF track_table[i_End].TAIoffset<>0 THEN
				 i_End:=F_I_number(i_End+1);
			  END_IF
			  track_table[i_End].TAIoffset:=TaiOffset[index];
			  track_table[i_End].Azimuth:= Azimuth[index];
			  track_table[i_End].Elevation:= Elevation[index];
		    END_FOR            
		   CommandArbiter.Status.LastLoadMode:= LoadMode; 
	       
		2:  i_Start:=1;       // Reset to 1st position of the stack. 
            i_End:= i_Start;  // Set the end of the table to the Start to over write the points. 
		                        // Consider adding a blend between the different tables. 
			FOR index:= ValidStart TO SequenceLength BY 1 DO  //New 
			  IF track_table[i_End].TAIoffset<>0 THEN
				 i_End:=F_I_number(i_End+1);
			  END_IF
			  track_table[i_End].TAIoffset:=TaiOffset[index];
			  track_table[i_End].Azimuth:= Azimuth[index];
			  track_table[i_End].Elevation:= Elevation[index];
		    END_FOR            
	           
	END_CASE;
	TrackLoadTable:= CmdResponseType.CommandActivated; // Reset
	CommandArbiter.Status.LastLoadMode:=LoadMode; 
	Tracking.TableStatus.pts_DataValid:=TRUE;
END_IF;

CommandArbiter.Status.LastCmdResponse:= TrackLoadTable;
END_METHOD

METHOD TrackStart :Uint
VAR_INPUT
	SessionID:UINT;
	Interpol:UINT;
	StartTime:LREAL;
END_VAR
VAR_OUTPUT
	
END_VAR
VAR
	
END_VAR
CASE CommandArbiter.Status.DscCmdAuthority OF                    // Check that corerct user is issueing a command
	LMC: IF SessionID= CommandArbiter.Lmc_ID THEN
			TrackStart:= CmdResponseType.CommandActivated;
     	 END_IF
			
	EGUI: IF SessionID= CommandArbiter.Egui_ID THEN
			TrackStart:= CmdResponseType.CommandActivated;
    	  END_IF		
ELSE 
     TrackStart:= CmdResponseType.NoCmdAuth;
     Command_Arbiter_error:=1;	
END_CASE

IF TrackStart = CmdResponseType.CommandActivated THEN // Dish State to see if move is possible
	Command_Arbiter_error:=0;
	IF  Management.ErrorStatus.errGeneral=0 AND Management.WarningStatus.waMngmnt =0 THEN  (*The Dish in the standby state*)
		CASE Management.Status.DscState OF 
			 DscStateType.Locked:        TrackStart:=CmdResponseType.DishLocked;
			 DscStateType.Locked_Stowed: TrackStart:=CmdResponseType.DishLocked;
			 DscStateType.Standstill:    TrackStart:=CmdResponseType.CommandActivated;
		     DscStateType.Standby:       TrackStart:=CmdResponseType.CommandActivated;
			 DscStateType.Stowed:	     TrackStart:=CmdResponseType.Stowed;
			 DscStateType.Track:         TrackStart:=CmdResponseType.CommandActivated;
		ELSE
		     TrackStart:=CmdResponseType.CommandRejected;
		     Command_Arbiter_error:=1;
		END_CASE								
	ELSE
		TrackStart:=CmdResponseType.CommandRejected;
		Command_Arbiter_error:=1;
	END_IF
END_IF
	
IF TrackStart=CmdResponseType.CommandActivated THEN
	IF StartTime > Time_cds.Status.TAIoffset THEN
		b_activate_Az:=1;
		b_activate_El:=1;	
		b_track_start:=1;
		lr_track_start_time:=StartTime;
	ELSIF StartTime < Time_cds.Status.TAIoffset THEN  // Will start tracking immediately
		b_activate_Az:=1;
		b_activate_El:=1;	
		b_track_start:=1;
		lr_track_start_time:=Time_cds.Status.TAIoffset;
	ELSIF StartTime < 0 THEN 
		TrackStart:=CmdResponseType.ParameterOutOfRange;
	ELSE 	
	//	TrackStart:=CmdResponseType.CommandActivated;
	//	b_activate_Az:=1;
	//	b_activate_El:=1;	
    //b_track_start:=1;
	//	lr_track_start_time:=Time_cds.Status.TAIoffset+0.1; // add 100ms to give enough time to start track. 
	END_IF			   
END_IF

Tracking.TableStatus.pts_Interpol:= Interpol;
CommandArbiter.Status.LastCmdResponse:=TrackStart;
END_METHOD

METHOD TrackStartPoly : UINT

VAR_INPUT
	SessionID:UINT;
	TrackId:  UINT;
	Order : UINT;
END_VAR

VAR
	
END_VAR
// Check Auth
// Check parameters
// Check State
TrackStartPoly := CmdResponseType.NotImplemented;

CommandArbiter.Status.LastCmdResponse:=TrackStartPoly;
END_METHOD

END_FUNCTION_BLOCK

// IndraMotionMlc1/Application/POUs/OPCUA/OPCUA_Node/P_Opcua_Management
PROGRAM P_Opcua_Management
VAR
	R_total_distance_AZ_old:LREAL;
	R_total_distance_EL_deg_old:LREAL;
	R_total_distance_EL_m_old:LREAL;
	R_total_distance_FI_old:LREAL;
	count_i:UINT;
	(*<<<<<<<<<<<<<<<<<<<<<<<<<<<<<<<<<<<< Stop >>>>>>>>>>>>>>>>>>>>>>>>>>>>>*)
	b_stop_Az_done: BOOL;
	b_stop_El_done: BOOL;
	b_stop_Fi_done: BOOL;
	fb_stop_Az: MC_Stop;
	fb_stop_El: MC_Stop;
	fb_stop_Fi: MC_Stop;
	rtrig_stop_Az: R_TRIG;
	rtrig_stop_El: R_TRIG;
	rtrig_stop_Fi: R_TRIG;
	rtrig_stop_stow: R_TRIG;
	rtrig_reset_stop: R_TRIG;
	
	(*<<<<<<<<<<<<<<<<<<<<<<<<<<<<<<<<<<<< Goto >>>>>>>>>>>>>>>>>>>>>>>>>>>>>*)
	// Az
	
	b_goto_done_Az: BOOL;
	b_active_Az:     BOOL;
	b_moving_Az: BOOL;
	fb_goto_Az: MC_MoveRelative;
	fb_start_goto_Az: R_Trig;
	fb_goto_done_Az : R_Trig;
	
	// El
	
	b_goto_done_El: BOOL;
	b_active_El:     BOOL;
	b_moving_El: BOOL;
	fb_goto_El: MC_MoveRelative;
	fb_start_goto_El: R_Trig;
	fb_goto_done_El : R_Trig;
	//Fi
	b_goto_done_Fi: BOOL;
	b_active_Fi:     BOOL;
	b_moving_Fi: BOOL;
	fb_goto_Fi: MC_MoveRelative;
	fb_start_goto_Fi: R_Trig;
	fb_goto_done_Fi : R_Trig;
	
(*<<<<<<<<<<<<<<<<<<<<<<<<<<<<<<<<<<<<<<<<<<<<<<<<<<<power>>>>>>>>>>>>>>>>>>>>>>>>>>>>>>>>>>>>*)
	ton_pow_off_Az: TON;
	ton_pow_off_El: TON;
	ton_pow_off_Fi: TON;
	rtrig_power_Az: R_TRIG;
	rtrig_power_El: R_TRIG;
	rtrig_power_Fi: R_TRIG;
	fb_ton_El: TON;
	fb_ton_Fi: TON;
	rtrig_off_Az: R_TRIG;
	rtrig_off_El: R_TRIG;
	rtrig_off_Fi: R_TRIG;
	rtrig_power_power: R_TRIG;
	b_pwr_on:BOOL;
	b_pwr_off: BOOL;
	b_clear_off_done_Az1: BOOL;
	b_clear_off_done_Az2: BOOL;
	b_clear_off_done_El: BOOL;
	b_clear_off_done_Fi1: BOOL;
	b_clear_off_done_Fi2: BOOL;
	
	FB_clear_error_off_Az1:MB_WriteParameter;
	FB_clear_error_off_Az2:MB_WriteParameter;
	FB_clear_error_off_El:MB_WriteParameter;
	FB_clear_error_off_Fi1:MB_WriteParameter;
	FB_clear_error_off_Fi2:MB_WriteParameter;
	rtrig_err: R_TRIG;
	rtrig_clear_done: R_TRIG;
	fb_ton_stow: TON;
	
	fb_rtrig_stow_deactivate1: R_TRIG;
	fb_rtrig_stow_deactivate: R_TRIG;
	b_execute_goto_Az: BOOL;
	R_TRIG_0: R_TRIG;
	R_TRIG_1: R_TRIG;
	rtrig_stop_goto_el: R_TRIG;
	rtrig_stop_goto_az: R_TRIG;
	fb_TON_2: TON;
	fb_TON_1: TON;
	r_goto_Az_rel: REAL;
	r_goto_El_rel: LREAL;
	r_goto_fi_rel: LREAL;
	fb_ton_stow1: TON;
END_VAR
VAR // added by the converter: edge detectors and wires of the graphical bodies
    _w1, _w2 : BOOL;
END_VAR


(***********Management.DscState***********)
IF azimuth.Status.AxisState=axisstatetype.StartUp OR elevation.Status.AxisState=axisstatetype.StartUp THEN
	Management.Status.DscState:=DscstateType.StartUp;
END_IF

IF azimuth.Status.AxisState=axisstatetype.Standby AND elevation.Status.AxisState=axisstatetype.Standby THEN
	Management.Status.DscState:=DscstateType.Standby;
END_IF

IF azimuth.Status.AxisState=axisstatetype.Activating OR elevation.Status.AxisState=axisstatetype.Activating THEN
	Management.Status.DscState:=DscstateType.Activating;
END_IF

IF azimuth.Status.AxisState=axisstatetype.Deactivating OR elevation.Status.AxisState=axisstatetype.Deactivating THEN
	Management.Status.DscState:=DscstateType.Deactivating;
END_IF

IF azimuth.Status.AxisState=axisstatetype.Standstill OR elevation.Status.AxisState=axisstatetype.Standstill THEN
	Management.Status.DscState:=DscstateType.Standstill;
END_IF

IF azimuth.Status.AxisState=axisstatetype.Stopping OR elevation.Status.AxisState=axisstatetype.Stopping THEN
	Management.Status.DscState:=DscstateType.stopping;
END_IF

IF azimuth.Status.AxisState=axisstatetype.Jog OR elevation.Status.AxisState=axisstatetype.Jog THEN
	Management.Status.DscState:=DscstateType.Jog;
END_IF

IF azimuth.Status.AxisState=axisstatetype.Slew OR elevation.Status.AxisState=axisstatetype.Slew THEN //capitalise S in slew
	Management.Status.DscState:=DscstateType.slew;
END_IF

IF azimuth.Status.AxisState=axisstatetype.Track AND elevation.Status.AxisState=axisstatetype.Track THEN
	Management.Status.DscState:=DscstateType.Track;
END_IF

IF azimuth.Status.AxisState=axisstatetype.Stowed THEN
	Management.Status.DscState:=DscstateType.Stowed;
END_IF
IF azimuth.Status.AxisState=axisstatetype.Locked OR elevation.Status.AxisState=axisstatetype.Locked THEN
	Management.Status.DscState:=DscstateType.Locked;
END_IF

IF azimuth.Status.AxisState=axisstatetype.Locked_Stowed OR elevation.Status.AxisState=axisstatetype.Locked_Stowed THEN
	Management.Status.DscState:=DscstateType.Locked_Stowed;
END_IF

// This one isn't going to work 
IF b_stow_pin_limit_lock AND (azimuth.Status.AxisState=axisstatetype.Locked OR elevation.Status.AxisState=axisstatetype.Locked) THEN     // Need to check Errors and interlocks to go into locked
	Management.Status.DscState:=DscstateType.Locked_Stowed;
END_IF

(*IF b_in_Estop THEN
	Management.Status.DscState:=DscstateType.Locked;  //Axis also need to go into locked state
END_IF
*)


// Work out where FiPOS is 
IF b_goto_done_Fi THEN 
	IF r_pos_fi_v < gc_r_band_optical+gc_r_band_tolerance AND r_pos_fi_v > gc_r_band_optical-gc_r_band_tolerance THEN 
		Management.Status.FiPos:= bandtype.Optical;
	ELSIF
		r_pos_fi_v < gc_r_band_1+gc_r_band_tolerance AND r_pos_fi_v > gc_r_band_1-gc_r_band_tolerance THEN 
		Management.Status.FiPos:= bandtype.Band_1;
	ELSIF
		r_pos_fi_v < gc_r_band_2+gc_r_band_tolerance AND r_pos_fi_v > gc_r_band_2-gc_r_band_tolerance THEN 
		Management.Status.FiPos:= bandtype.Band_2;
	ELSIF
		r_pos_fi_v < gc_r_band_3+gc_r_band_tolerance AND r_pos_fi_v > gc_r_band_3-gc_r_band_tolerance THEN 
		Management.Status.FiPos:= bandtype.Band_3;
	ELSIF
		r_pos_fi_v < gc_r_band_4+gc_r_band_tolerance AND r_pos_fi_v > gc_r_band_4-gc_r_band_tolerance THEN 
		Management.Status.FiPos:= bandtype.Band_4;
	ELSIF
		r_pos_fi_v < gc_r_band_5a+gc_r_band_tolerance AND r_pos_fi_v > gc_r_band_5a-gc_r_band_tolerance THEN 
		Management.Status.FiPos:= bandtype.Band_5a;
	ELSIF
		r_pos_fi_v < gc_r_band_5b+gc_r_band_tolerance AND r_pos_fi_v > gc_r_band_5b-gc_r_band_tolerance THEN 
		Management.Status.FiPos:= bandtype.Band_5b;
	ELSIF
		r_pos_fi_v < gc_r_band_6+gc_r_band_tolerance AND r_pos_fi_v > gc_r_band_6-gc_r_band_tolerance THEN 
		Management.Status.FiPos:= bandtype.Band_6;
	ELSE
		Management.Status.FiPos:= bandtype.Unknown;
	END_IF

END_IF


//Management.Status.FiPos:=Current_FIPos; // this needs to be of band type 
Management.Status.HHP_Cncted:=b_HHP_Connected;
Management.Status.HHP_Az:=b_HHP_AZ;
Management.Status.HHP_El:=b_HHP_EL;
IF b_HHP_AZ = FALSE AND b_HHP_EL= FALSE THEN
	Management.Status.HHP_Fi:=TRUE;
ELSE
	Management.Status.HHP_Fi:=FALSE;
END_IF
IF b_HHP_move_cw_slow OR b_HHP_move_cw_fast THEN
	Management.Status.HHP_Dir_Plus	:= TRUE;
ELSE
	Management.Status.HHP_Dir_Plus	:= FALSE;
END_IF
IF b_HHP_move_ccw_slow OR b_HHP_move_ccw_fast THEN
	Management.Status.HHP_Dir_Minus:= TRUE;
ELSE
	Management.Status.HHP_Dir_Minus:= FALSE;
END_IF

(*********NamePlate**********)
Management.NamePlate.RunHours:=r_operation_hour;

count_i:=count_i+1;
IF count_i = 5 THEN
	R_total_distance_AZ:=ABS(r_pos_az-R_total_distance_AZ_old)+R_total_distance_AZ;
	R_total_distance_AZ_old:=r_pos_az;
	R_total_distance_EL_deg:=ABS(r_pos_el-R_total_distance_el_deg_old)+R_total_distance_el_deg;
	R_total_distance_EL_m:=R_total_distance_EL_deg/K_gear_ratio;
	R_total_distance_el_deg_old:=r_pos_el;
	R_total_distance_FI:=ABS(r_pos_FI-R_total_distance_FI_old)+R_total_distance_FI;
	R_total_distance_FI_old:=r_pos_FI;
	count_i:=0;
END_IF

Management.NamePlate.TotalDist_Az:=R_total_distance_AZ;
Management.NamePlate.TotalDist_El_deg:=R_total_distance_EL_deg;
Management.NamePlate.TotalDist_El_m:=R_total_distance_EL_m;
Management.NamePlate.TotalDist_Fi:=R_total_distance_FI;

(*********TempHumidStatus**********)
Management.TempHumidStatus.HumidDriveCab:=LREAL_TO_REAL(HumidDriveCab);
Management.TempHumidStatus.TempDriveCab:=LREAL_TO_REAL(TempDriveCab);
Management.TempHumidStatus.HumidPSC_Inlet:=LREAL_TO_REAL(HumidPSC_Inlet);
Management.TempHumidStatus.TempPSC_Inlet:=LREAL_TO_REAL(TempPSC_Inlet);
Management.TempHumidStatus.HumidPSC_Outlet:=LREAL_TO_REAL(HumidPSC_Outlet);
Management.TempHumidStatus.TempPSC_Outlet:=LREAL_TO_REAL(TempPSC_Outlet);
Management.TempHumidStatus.TempEMISC_Outlet:=LREAL_TO_REAL(TempEMISC_Outlet);

(*********PowerStatus**********)
Management.PowerStatus.cbEMISC:=b_PSC_PD_EMISC_Breaker_on;
Management.PowerStatus.cbFan_PSC:=b_PSC_PD_FAN_Breaker_on;
Management.PowerStatus.cbPSC_Spare:=b_PSC_PD_spare;
Management.PowerStatus.cbHe_Comp:=b_MAIN_PD_Compressor_breaker_on;
Management.PowerStatus.cbPDU_Fi:=b_MAIN_PD_FI_Breaker_on;
Management.PowerStatus.cbPED_Spare:=b_MAIN_PD_spare;
Management.PowerStatus.ActPwrCnsm:= 0; // Needs to be updated with real number
Management.PowerStatus.CurrentPh1:= LREAL_TO_REAL(CurrentPh1);
Management.PowerStatus.CurrentPh2:=LREAL_TO_REAL(CurrentPh2);
Management.PowerStatus.CurrentPh3:=LREAL_TO_REAL(CurrentPh3);
Management.PowerStatus.FrequencyPh1:=LREAL_TO_REAL(FrequencyPh1);
Management.PowerStatus.FrequencyPh2:=LREAL_TO_REAL(FrequencyPh2);
Management.PowerStatus.FrequencyPh3:=LREAL_TO_REAL(FrequencyPh3);
Management.PowerStatus.VoltagePh1:=LREAL_TO_REAL(VoltagePh1);
Management.PowerStatus.VoltagePh2:=LREAL_TO_REAL(VoltagePh2);
Management.PowerStatus.VoltagePh3:=LREAL_TO_REAL(VoltagePh3);
Management.PowerStatus.PowerFactor:=LREAL_TO_REAL(PowerFactor);
//Management.PowerStatus.LowPowerActive:=0;  

(*********ErrorStatus**********)

//Management.ErrorStatus.errAuthLost:=0;
Management.ErrorStatus.errAzimuth:=(axisdata[1].Axis_Error OR axisdata[2].Axis_Error);  
Management.ErrorStatus.errElevation:=(axisdata[3].Axis_Error);  
Management.ErrorStatus.errFeedindexer:=(axisdata[4].Axis_Error OR axisdata[5].Axis_Error); 
Management.ErrorStatus.errPoint:=0;
IF safety.Status.SafetyState=0 THEN
	Management.ErrorStatus.errSafety:=0;
ELSE
	Management.ErrorStatus.errSafety:=1;
END_IF
Management.ErrorStatus.errTime:=axisdata[10].Axis_Error;
Management.ErrorStatus.errCmd:=Command_Arbiter_error;
Management.ErrorStatus.errTrack:=(NOT(tracking.Status.tr_initOk) AND b_track_on);
Management.ErrorStatus.errStwPin:=NOT((b_stow_pin_limit_lock XOR b_stow_pin_limit_unlock)XOR(b_stow_pin_retract XOR b_stow_pin_deploy));
IF status_code1 = 'F8070' OR status_code2 = 'F8070' OR status_code3 = 'F8070' OR status_code4 = 'F8070' OR status_code5 = 'F8070' THEN
	Management.ErrorStatus.errPwr24VDC:=1;
ELSE
	Management.ErrorStatus.errPwr24VDC:=0;
END_IF
IF status_code1 = 'F2802' OR status_code2 = 'F2802' OR status_code3 = 'F2802' OR status_code4 = 'F2802' OR status_code5 = 'F2802' THEN
	Management.ErrorStatus.errPwr400VAC:=1;
ELSE
	Management.ErrorStatus.errPwr400VAC:=0;
END_IF
IF status_code1 = 'F2802' OR status_code2 = 'F2802' OR status_code3 = 'F2802' OR status_code4 = 'F2802' OR status_code5 = 'F2802' THEN
	Management.ErrorStatus.errPwr400VAC:=1;
ELSE
	Management.ErrorStatus.errPwr400VAC:=0;
END_IF
IF status_code1 = 'F8091' OR status_code2 = 'F8091' OR status_code3 = 'F8091' OR status_code4 = 'F8091' OR status_code5 = 'F8091' THEN
	Management.ErrorStatus.errPwr400VAC:=1;
ELSE
	Management.ErrorStatus.errPwr400VAC:=0;
END_IF
//	Management.ErrorStatus.errPwrMeterComms:=0;
//	Management.ErrorStatus.errTiltOneComms:=0;
//	Management.ErrorStatus.errTiltOneIoUnit:=0;
//	Management.ErrorStatus.errTiltTwoComms:=0;
//	Management.ErrorStatus.errTiltTwoIoUnit:=0;

Management.ErrorStatus.errGeneral:=(Management.ErrorStatus.errAzimuth OR Management.ErrorStatus.errElevation OR Management.ErrorStatus.errFeedindexer OR Management.ErrorStatus.errSafety OR Management.ErrorStatus.errTime OR Management.ErrorStatus.errTrack OR Management.ErrorStatus.errPoint);
Management.ErrorStatus.errMngmnt:=Management.ErrorStatus.errGeneral;

(*********WarningStatus**********)
//IF gc_b_sim_on = 0 THEN 
	Management.WarningStatus.waAzimuth:=(axisdata[1].Axis_Warning OR axisdata[2].Axis_Warning);
    Management.WarningStatus.waElevation:=(axisdata[3].Axis_Warning);
    Management.WarningStatus.waFeedindexer:=(axisdata[4].Axis_Warning OR axisdata[5].Axis_Warning);
//ELSIF gc_b_sim_on =1 THEN
//	Management.WarningStatus.waAzimuth:=(

Management.WarningStatus.waCmd:=0;
Management.WarningStatus.waPoint:=0;
Management.WarningStatus.waSafety:=0;
Management.WarningStatus.waStwPin:=0;
Management.WarningStatus.waPoint:=0;
Management.WarningStatus.waTime:=0;
Management.WarningStatus.waTrack:=0;
Management.WarningStatus.waDoorDrive:=b_DriveCabinetDoor_Estop;
Management.WarningStatus.waDoorEMISC:=b_EMISCDoor_Estop;
Management.WarningStatus.waDoorPED:=b_DSDoor_Estop;
Management.WarningStatus.waDoorPSC:=b_PSCDoor_Estop;
Management.WarningStatus.waHatchPscRoof:=0;
Management.WarningStatus.waHatchAzBearing:=b_AZ_Hatch;
Management.WarningStatus.waHornOn:=b_Horn;
//Management.WarningStatus.waOverTempDrive
//Management.WarningStatus.waOverTempEMISC
//Management.WarningStatus.waDoorPED
//Management.WarningStatus.waDoorPSC
Management.WarningStatus.waSafe2ApproachLight:=0;

// Power mode control 
// Need to limit velocity and acceleration to keep the power below the limit 


// Run Ladder logic
P_Opcua_Management.A_CLR_ERR();
P_Opcua_Management.A_STOP();
P_Opcua_Management.A_GOTO();

ACTION A_CLR_ERR:
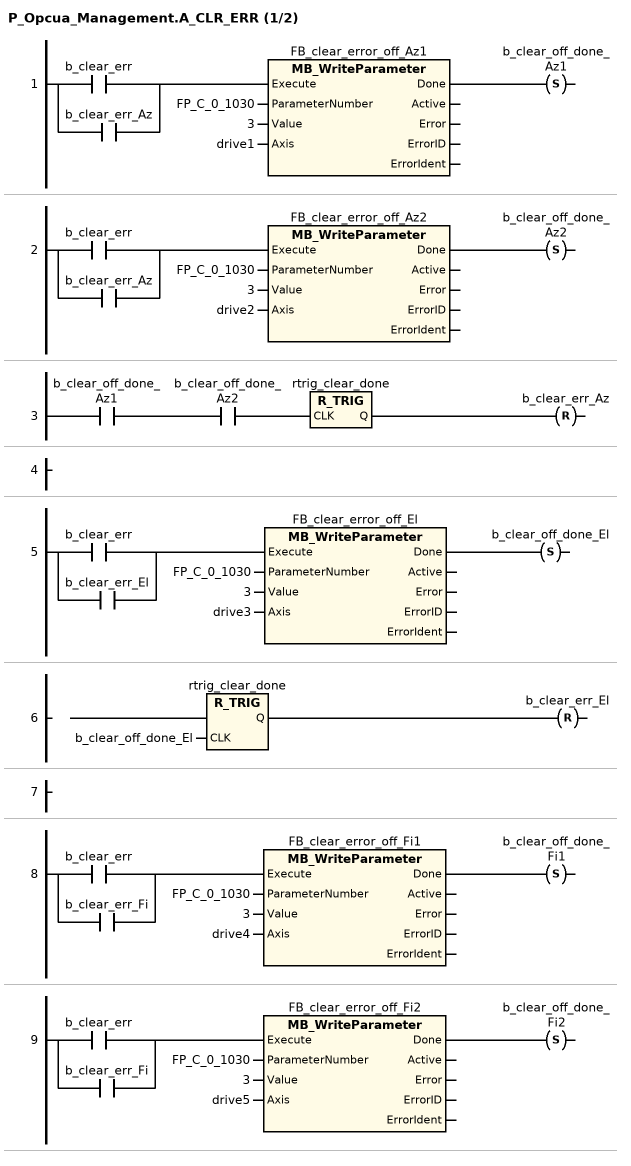
// NETWORK 1
//   FP_C_0_1030: Command: Clear all control errors
//   drive1: Real axis "Drive1" with axis number 1
FB_clear_error_off_Az1(
    Execute := b_clear_err OR b_clear_err_Az,
    ParameterNumber := FP_C_0_1030,
    Value := 3,
    Axis := drive1); // MB_WriteParameter
b_clear_off_done_Az1 S= FB_clear_error_off_Az1.Done;

// NETWORK 2
//   FP_C_0_1030: Command: Clear all control errors
//   drive2: Real axis "Drive1" with axis number 1
FB_clear_error_off_Az2(
    Execute := b_clear_err OR b_clear_err_Az,
    ParameterNumber := FP_C_0_1030,
    Value := 3,
    Axis := drive2); // MB_WriteParameter
b_clear_off_done_Az2 S= FB_clear_error_off_Az2.Done;

// NETWORK 3
rtrig_clear_done(CLK := b_clear_off_done_Az1 AND b_clear_off_done_Az2); // R_TRIG
b_clear_err_Az R= rtrig_clear_done.Q;

// NETWORK 4

// NETWORK 5
//   FP_C_0_1030: Command: Clear all control errors
//   drive3: Real axis "Drive1" with axis number 1
FB_clear_error_off_El(
    Execute := b_clear_err OR b_clear_err_El,
    ParameterNumber := FP_C_0_1030,
    Value := 3,
    Axis := drive3); // MB_WriteParameter
b_clear_off_done_El S= FB_clear_error_off_El.Done;

// NETWORK 6
rtrig_clear_done(CLK := b_clear_off_done_El); // R_TRIG
b_clear_err_El R= rtrig_clear_done.Q;

// NETWORK 7

// NETWORK 8
//   FP_C_0_1030: Command: Clear all control errors
//   drive4: Real axis "Drive1" with axis number 1
FB_clear_error_off_Fi1(
    Execute := b_clear_err OR b_clear_err_Fi,
    ParameterNumber := FP_C_0_1030,
    Value := 3,
    Axis := drive4); // MB_WriteParameter
b_clear_off_done_Fi1 S= FB_clear_error_off_Fi1.Done;

// NETWORK 9
//   FP_C_0_1030: Command: Clear all control errors
//   drive5: Real axis "Drive1" with axis number 1
FB_clear_error_off_Fi2(
    Execute := b_clear_err OR b_clear_err_Fi,
    ParameterNumber := FP_C_0_1030,
    Value := 3,
    Axis := drive5); // MB_WriteParameter
b_clear_off_done_Fi2 S= FB_clear_error_off_Fi2.Done;

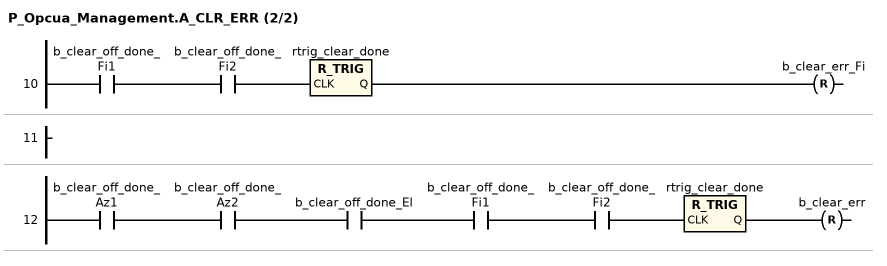
// NETWORK 10
rtrig_clear_done(CLK := b_clear_off_done_Fi1 AND b_clear_off_done_Fi2); // R_TRIG
b_clear_err_Fi R= rtrig_clear_done.Q;

// NETWORK 11

// NETWORK 12
rtrig_clear_done(CLK := b_clear_off_done_Az1 AND b_clear_off_done_Az2 AND b_clear_off_done_El AND b_clear_off_done_Fi1 AND b_clear_off_done_Fi2); // R_TRIG
b_clear_err R= rtrig_clear_done.Q;
END_ACTION

ACTION A_GOTO:
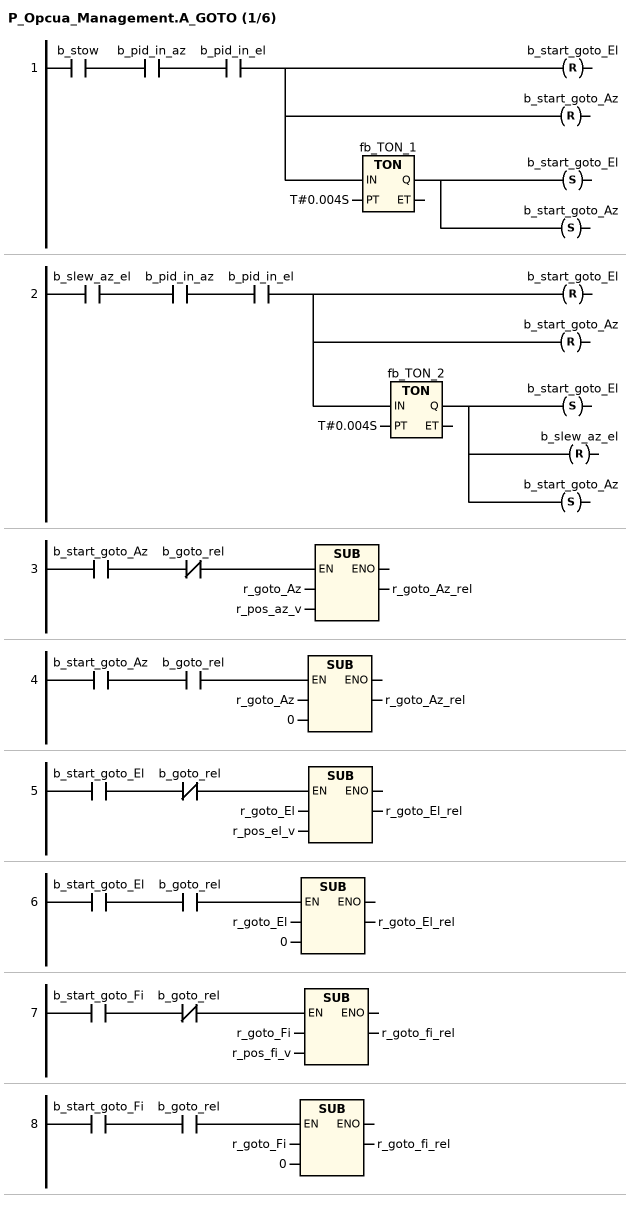
// NETWORK 1
_w1 := b_stow AND b_pid_in_az AND b_pid_in_el;
b_start_goto_El R= _w1;
b_start_goto_Az R= _w1;
fb_TON_1(IN := _w1, PT := T#0.004S); // TON
b_start_goto_El S= fb_TON_1.Q;
b_start_goto_Az S= fb_TON_1.Q;

// NETWORK 2
_w2 := b_slew_az_el AND b_pid_in_az AND b_pid_in_el;
b_start_goto_El R= _w2;
b_start_goto_Az R= _w2;
fb_TON_2(IN := _w2, PT := T#0.004S); // TON
b_start_goto_El S= fb_TON_2.Q;
b_slew_az_el R= fb_TON_2.Q;
b_start_goto_Az S= fb_TON_2.Q;

// NETWORK 3
IF b_start_goto_Az AND NOT b_goto_rel THEN r_goto_Az_rel := r_goto_Az - r_pos_az_v; END_IF

// NETWORK 4
IF b_start_goto_Az AND b_goto_rel THEN r_goto_Az_rel := r_goto_Az - 0; END_IF

// NETWORK 5
IF b_start_goto_El AND NOT b_goto_rel THEN r_goto_El_rel := r_goto_El - r_pos_el_v; END_IF

// NETWORK 6
IF b_start_goto_El AND b_goto_rel THEN r_goto_El_rel := r_goto_El - 0; END_IF

// NETWORK 7
IF b_start_goto_Fi AND NOT b_goto_rel THEN r_goto_fi_rel := r_goto_Fi - r_pos_fi_v; END_IF

// NETWORK 8
IF b_start_goto_Fi AND b_goto_rel THEN r_goto_fi_rel := r_goto_Fi - 0; END_IF

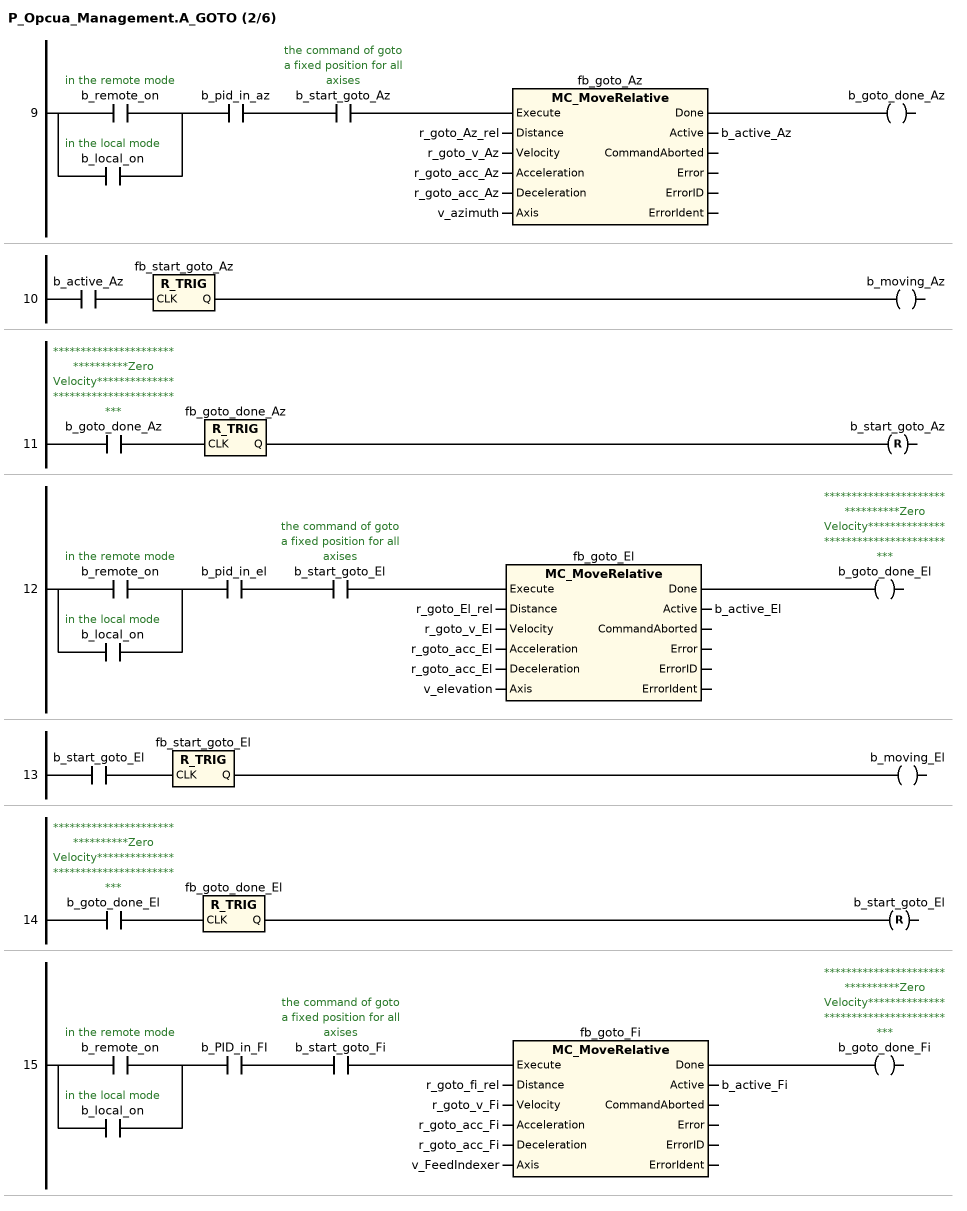
// NETWORK 9
//   b_remote_on: in the remote mode
//   b_local_on: in the local mode
//   b_start_goto_Az: the command of goto a fixed position for all axises
//   r_goto_Az_rel: actual value of goto
//   v_azimuth: Virtual axis "v_azimuth" with axis number 7
fb_goto_Az(
    Execute := (b_remote_on OR b_local_on) AND b_pid_in_az AND b_start_goto_Az,
    Distance := r_goto_Az_rel,
    Velocity := r_goto_v_Az,
    Acceleration := r_goto_acc_Az,
    Deceleration := r_goto_acc_Az,
    Axis := v_azimuth,
    Active => b_active_Az); // MC_MoveRelative
b_goto_done_Az := fb_goto_Az.Done;

// NETWORK 10
fb_start_goto_Az(CLK := b_active_Az); // R_TRIG
b_moving_Az := fb_start_goto_Az.Q;

// NETWORK 11
//   b_goto_done_Az: ********************************Zero Velocity***************************************
fb_goto_done_Az(CLK := b_goto_done_Az); // R_TRIG
b_start_goto_Az R= fb_goto_done_Az.Q;

// NETWORK 12
//   b_remote_on: in the remote mode
//   b_local_on: in the local mode
//   b_start_goto_El: the command of goto a fixed position for all axises
//   r_goto_El_rel: actual value of goto
//   v_elevation: Virtual axis "v_azimuth" with axis number 7
//   b_goto_done_El: ********************************Zero Velocity***************************************
fb_goto_El(
    Execute := (b_remote_on OR b_local_on) AND b_pid_in_el AND b_start_goto_El,
    Distance := r_goto_El_rel,
    Velocity := r_goto_v_El,
    Acceleration := r_goto_acc_El,
    Deceleration := r_goto_acc_El,
    Axis := v_elevation,
    Active => b_active_El); // MC_MoveRelative
b_goto_done_El := fb_goto_El.Done;

// NETWORK 13
fb_start_goto_El(CLK := b_start_goto_El); // R_TRIG
b_moving_El := fb_start_goto_El.Q;

// NETWORK 14
//   b_goto_done_El: ********************************Zero Velocity***************************************
fb_goto_done_El(CLK := b_goto_done_El); // R_TRIG
b_start_goto_El R= fb_goto_done_El.Q;

// NETWORK 15
//   b_remote_on: in the remote mode
//   b_local_on: in the local mode
//   b_start_goto_Fi: the command of goto a fixed position for all axises
//   r_goto_fi_rel: actual value of goto
//   v_FeedIndexer: Virtual axis "v_azimuth" with axis number 7
//   b_goto_done_Fi: ********************************Zero Velocity***************************************
fb_goto_Fi(
    Execute := (b_remote_on OR b_local_on) AND b_PID_in_FI AND b_start_goto_Fi,
    Distance := r_goto_fi_rel,
    Velocity := r_goto_v_Fi,
    Acceleration := r_goto_acc_Fi,
    Deceleration := r_goto_acc_Fi,
    Axis := v_FeedIndexer,
    Active => b_active_Fi); // MC_MoveRelative
b_goto_done_Fi := fb_goto_Fi.Done;

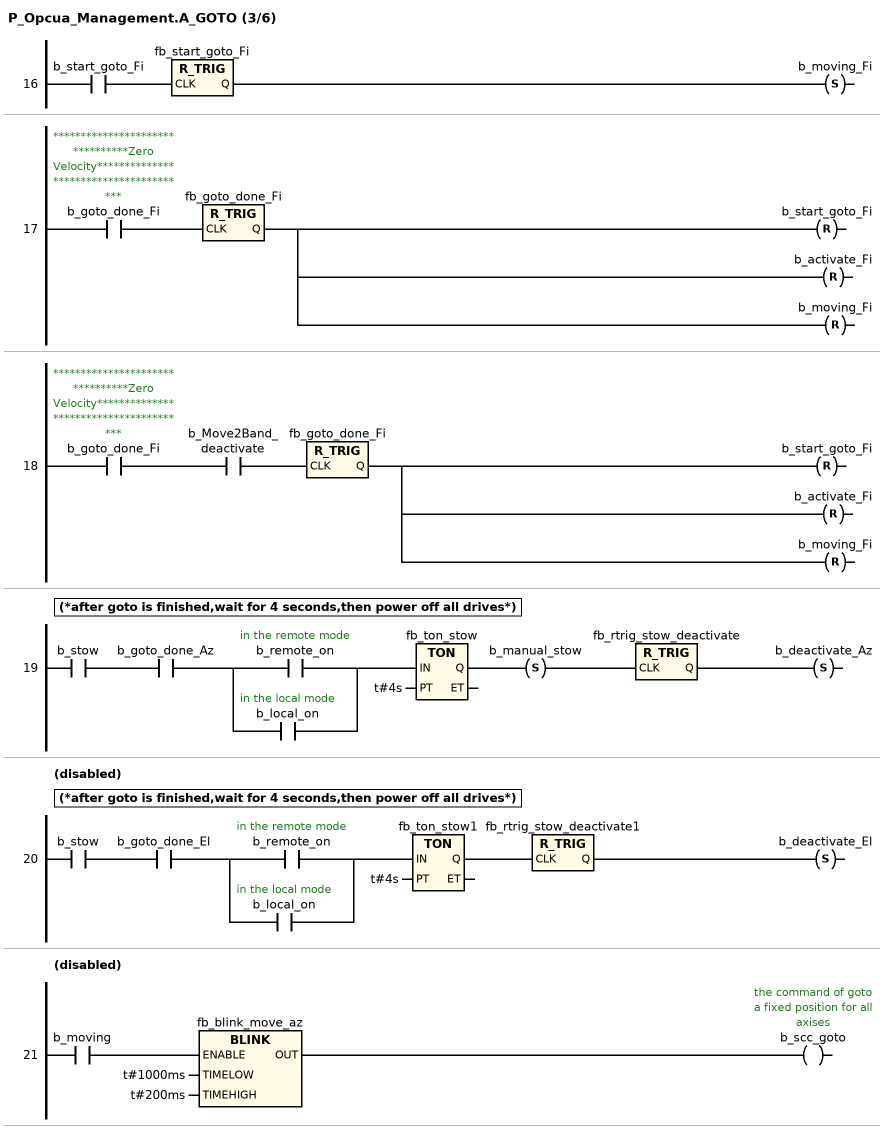
// NETWORK 16
fb_start_goto_Fi(CLK := b_start_goto_Fi); // R_TRIG
b_moving_Fi S= fb_start_goto_Fi.Q;

// NETWORK 17
//   b_goto_done_Fi: ********************************Zero Velocity***************************************
fb_goto_done_Fi(CLK := b_goto_done_Fi); // R_TRIG
b_start_goto_Fi R= fb_goto_done_Fi.Q;
b_activate_Fi R= fb_goto_done_Fi.Q;
b_moving_Fi R= fb_goto_done_Fi.Q;

// NETWORK 18
//   b_goto_done_Fi: ********************************Zero Velocity***************************************
fb_goto_done_Fi(CLK := b_goto_done_Fi AND b_Move2Band_deactivate); // R_TRIG
b_start_goto_Fi R= fb_goto_done_Fi.Q;
b_activate_Fi R= fb_goto_done_Fi.Q;
b_moving_Fi R= fb_goto_done_Fi.Q;

// NETWORK 19
//   fb_rtrig_stow_deactivate: the definition of rise trigger,The function block R_TRIG detects a rising edge.
//   fb_ton_stow: The function block Timer On Delay implements a turn-on delay
//   b_remote_on: in the remote mode
//   b_local_on: in the local mode
// label: (*after goto is finished,wait for 4 seconds,then power off all drives*)
fb_ton_stow(IN := b_stow AND b_goto_done_Az AND (b_remote_on OR b_local_on), PT := t#4s); // TON
b_manual_stow S= fb_ton_stow.Q;
fb_rtrig_stow_deactivate(CLK := fb_ton_stow.Q); // R_TRIG
b_deactivate_Az S= fb_rtrig_stow_deactivate.Q;

// NETWORK 20 (disabled)
//   fb_rtrig_stow_deactivate1: the definition of rise trigger,The function block R_TRIG detects a rising edge.
//   fb_ton_stow1: The function block Timer On Delay implements a turn-on delay
//   b_remote_on: in the remote mode
//   b_local_on: in the local mode
// label: (*after goto is finished,wait for 4 seconds,then power off all drives*)
// fb_ton_stow1(IN := b_stow AND b_goto_done_El AND (b_remote_on OR b_local_on), PT := t#4s); // TON
// fb_rtrig_stow_deactivate1(CLK := fb_ton_stow1.Q); // R_TRIG
// b_deactivate_El S= fb_rtrig_stow_deactivate1.Q;

// NETWORK 21 (disabled)
//   b_scc_goto: the command of goto a fixed position for all axises
// fb_blink_move_az(ENABLE := b_moving, TIMELOW := t#1000ms, TIMEHIGH := t#200ms); // BLINK
// b_scc_goto := fb_blink_move_az.OUT;

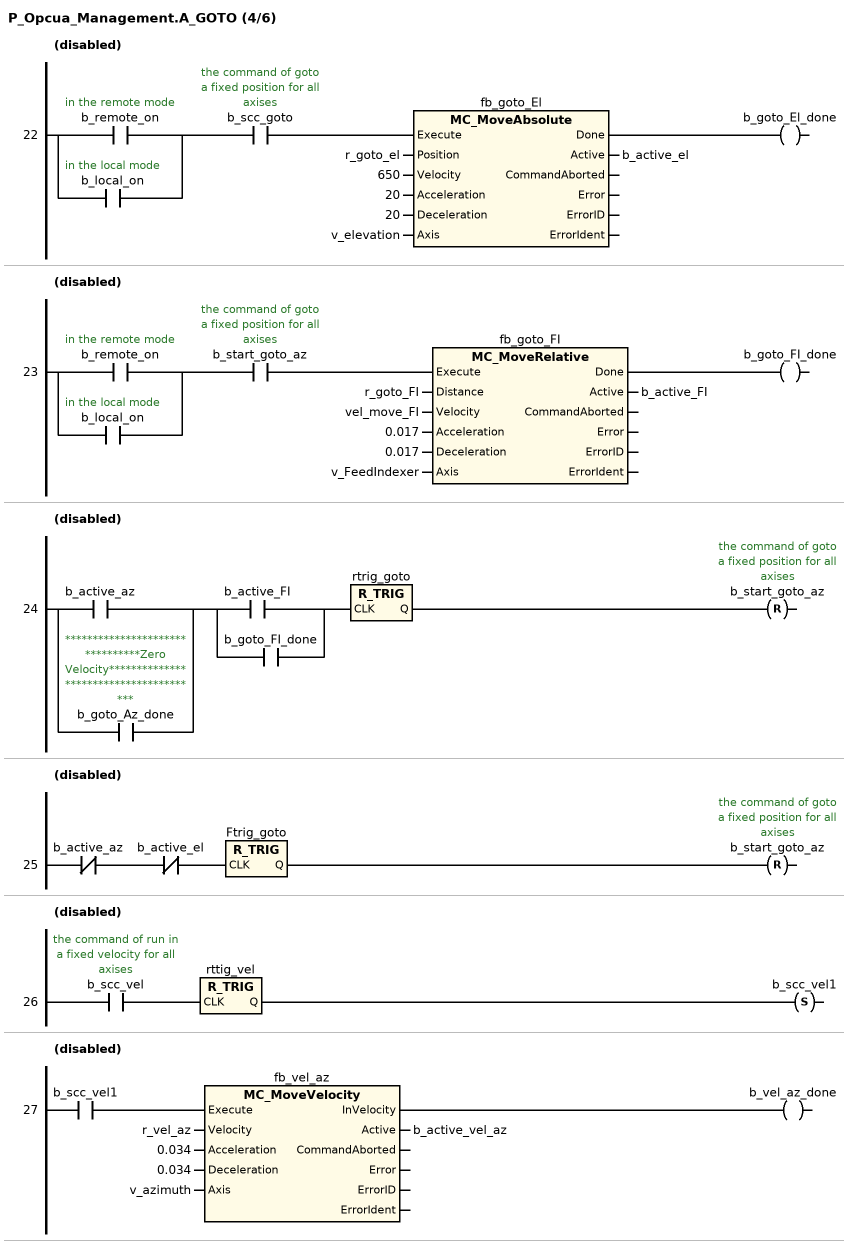
// NETWORK 22 (disabled)
//   b_remote_on: in the remote mode
//   b_local_on: in the local mode
//   b_scc_goto: the command of goto a fixed position for all axises
//   v_elevation: Virtual axis "v_elevation" with axis number 8
// fb_goto_El(
//     Execute := (b_remote_on OR b_local_on) AND b_scc_goto,
//     Position := r_goto_el,
//     Velocity := 650,
//     Acceleration := 20,
//     Deceleration := 20,
//     Axis := v_elevation,
//     Active => b_active_el); // MC_MoveAbsolute
// b_goto_El_done := fb_goto_El.Done;

// NETWORK 23 (disabled)
//   b_remote_on: in the remote mode
//   b_local_on: in the local mode
//   b_start_goto_az: the command of goto a fixed position for all axises
//   v_FeedIndexer: Virtual axis "v_polarization" with axis number 9
// fb_goto_FI(
//     Execute := (b_remote_on OR b_local_on) AND b_start_goto_az,
//     Distance := r_goto_FI,
//     Velocity := vel_move_FI,
//     Acceleration := 0.017,
//     Deceleration := 0.017,
//     Axis := v_FeedIndexer,
//     Active => b_active_FI); // MC_MoveRelative
// b_goto_FI_done := fb_goto_FI.Done;

// NETWORK 24 (disabled)
//   b_goto_Az_done: ********************************Zero Velocity***************************************
//   b_start_goto_az: the command of goto a fixed position for all axises
// rtrig_goto(CLK := (b_active_az OR b_goto_Az_done) AND (b_active_FI OR b_goto_FI_done)); // R_TRIG
// b_start_goto_az R= rtrig_goto.Q;

// NETWORK 25 (disabled)
//   b_start_goto_az: the command of goto a fixed position for all axises
// Ftrig_goto(CLK := NOT b_active_az AND NOT b_active_el); // R_TRIG
// b_start_goto_az R= Ftrig_goto.Q;

// NETWORK 26 (disabled)
//   b_scc_vel: the command of run in a fixed velocity for all axises
// rttig_vel(CLK := b_scc_vel); // R_TRIG
// b_scc_vel1 S= rttig_vel.Q;

// NETWORK 27 (disabled)
//   r_vel_az: ************vel*************
//   v_azimuth: Virtual axis "v_azimuth" with axis number 7
// fb_vel_az(
//     Execute := b_scc_vel1,
//     Velocity := r_vel_az,
//     Acceleration := 0.034,
//     Deceleration := 0.034,
//     Axis := v_azimuth,
//     Active => b_active_vel_az); // MC_MoveVelocity
// b_vel_az_done := fb_vel_az.InVelocity;

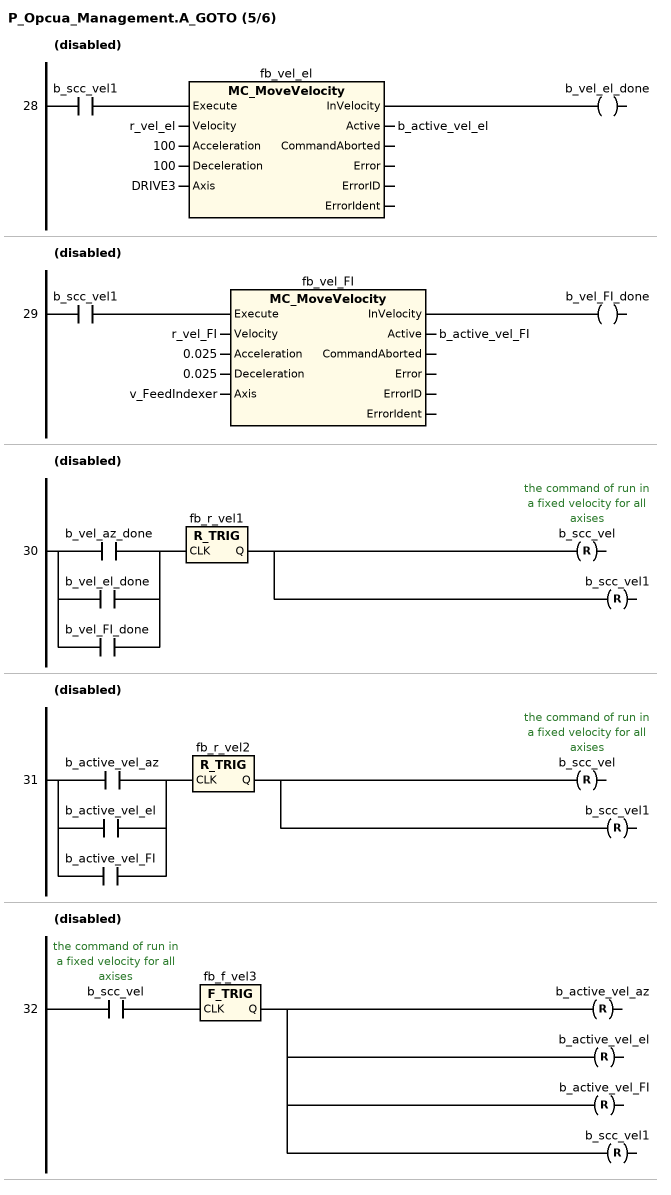
// NETWORK 28 (disabled)
//   DRIVE3: Virtual axis "v_elevation" with axis number 8
// fb_vel_el(
//     Execute := b_scc_vel1,
//     Velocity := r_vel_el,
//     Acceleration := 100,
//     Deceleration := 100,
//     Axis := DRIVE3,
//     Active => b_active_vel_el); // MC_MoveVelocity
// b_vel_el_done := fb_vel_el.InVelocity;

// NETWORK 29 (disabled)
//   v_FeedIndexer: Virtual axis "v_polarization" with axis number 9
// fb_vel_FI(
//     Execute := b_scc_vel1,
//     Velocity := r_vel_FI,
//     Acceleration := 0.025,
//     Deceleration := 0.025,
//     Axis := v_FeedIndexer,
//     Active => b_active_vel_FI); // MC_MoveVelocity
// b_vel_FI_done := fb_vel_FI.InVelocity;

// NETWORK 30 (disabled)
//   b_scc_vel: the command of run in a fixed velocity for all axises
// fb_r_vel1(CLK := b_vel_az_done OR b_vel_el_done OR b_vel_FI_done); // R_TRIG
// b_scc_vel R= fb_r_vel1.Q;
// b_scc_vel1 R= fb_r_vel1.Q;

// NETWORK 31 (disabled)
//   b_scc_vel: the command of run in a fixed velocity for all axises
// fb_r_vel2(CLK := b_active_vel_az OR b_active_vel_el OR b_active_vel_FI); // R_TRIG
// b_scc_vel R= fb_r_vel2.Q;
// b_scc_vel1 R= fb_r_vel2.Q;

// NETWORK 32 (disabled)
//   b_scc_vel: the command of run in a fixed velocity for all axises
// fb_f_vel3(CLK := b_scc_vel); // F_TRIG
// b_active_vel_az R= fb_f_vel3.Q;
// b_active_vel_el R= fb_f_vel3.Q;
// b_active_vel_FI R= fb_f_vel3.Q;
// b_scc_vel1 R= fb_f_vel3.Q;

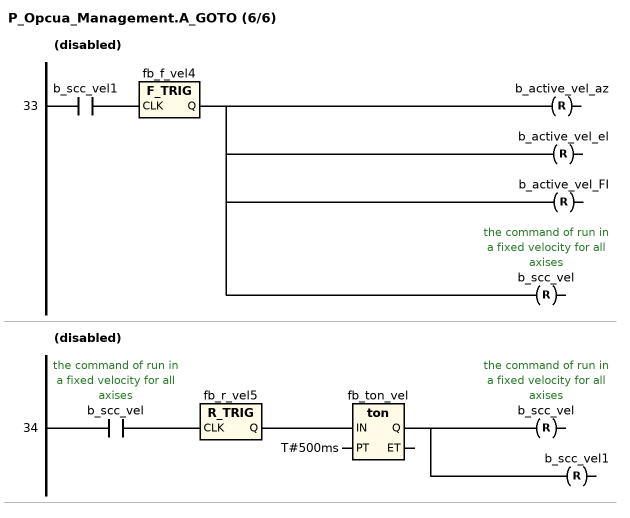
// NETWORK 33 (disabled)
//   b_scc_vel: the command of run in a fixed velocity for all axises
// fb_f_vel4(CLK := b_scc_vel1); // F_TRIG
// b_active_vel_az R= fb_f_vel4.Q;
// b_active_vel_el R= fb_f_vel4.Q;
// b_active_vel_FI R= fb_f_vel4.Q;
// b_scc_vel R= fb_f_vel4.Q;

// NETWORK 34 (disabled)
//   b_scc_vel: the command of run in a fixed velocity for all axises
// fb_r_vel5(CLK := b_scc_vel); // R_TRIG
// fb_ton_vel(IN := fb_r_vel5.Q, PT := T#500ms); // ton
// b_scc_vel R= fb_ton_vel.Q;
// b_scc_vel1 R= fb_ton_vel.Q;
END_ACTION

ACTION A_STOP:
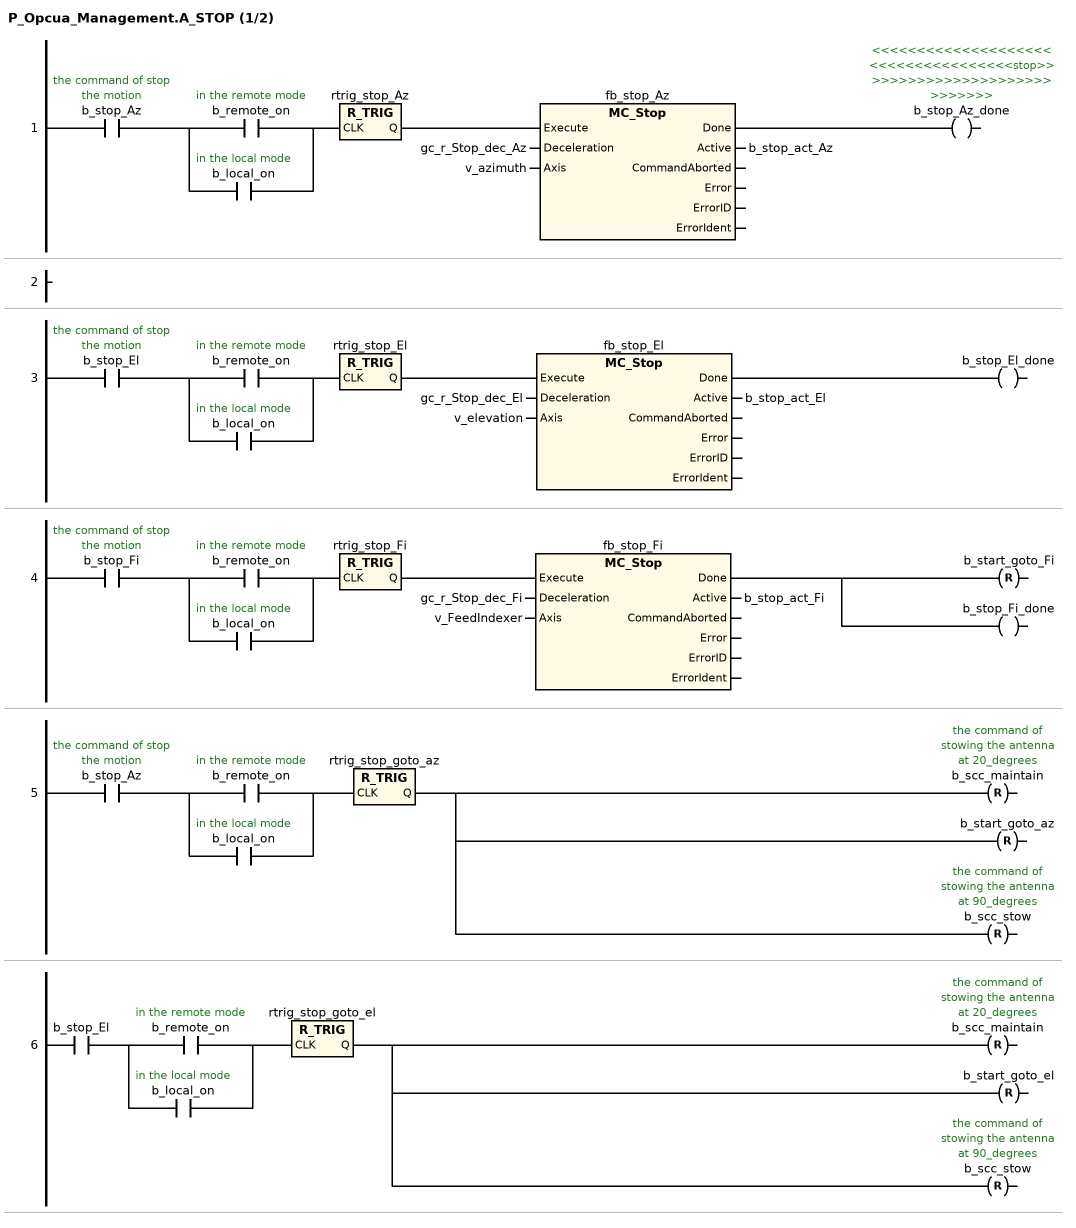
// NETWORK 1
//   b_stop_Az: the command of stop the motion
//   b_remote_on: in the remote mode
//   b_local_on: in the local mode
//   v_azimuth: Virtual axis "v_azimuth" with axis number 7
//   b_stop_Az_done: <<<<<<<<<<<<<<<<<<<<<<<<<<<<<<<<<<<<stop>>>>>>>>>>>>>>>>>>>>>>>>>>>>>
rtrig_stop_Az(CLK := b_stop_Az AND (b_remote_on OR b_local_on)); // R_TRIG
fb_stop_Az(
    Execute := rtrig_stop_Az.Q,
    Deceleration := gc_r_Stop_dec_Az,
    Axis := v_azimuth,
    Active => b_stop_act_Az); // MC_Stop
b_stop_Az_done := fb_stop_Az.Done;

// NETWORK 2

// NETWORK 3
//   b_stop_El: the command of stop the motion
//   b_remote_on: in the remote mode
//   b_local_on: in the local mode
//   v_elevation: Virtual axis "v_elevation" with axis number 8
rtrig_stop_El(CLK := b_stop_El AND (b_remote_on OR b_local_on)); // R_TRIG
fb_stop_El(
    Execute := rtrig_stop_El.Q,
    Deceleration := gc_r_Stop_dec_El,
    Axis := v_elevation,
    Active => b_stop_act_El); // MC_Stop
b_stop_El_done := fb_stop_El.Done;

// NETWORK 4
//   b_stop_Fi: the command of stop the motion
//   b_remote_on: in the remote mode
//   b_local_on: in the local mode
//   v_FeedIndexer: Virtual axis "v_polarization" with axis number 9
rtrig_stop_Fi(CLK := b_stop_Fi AND (b_remote_on OR b_local_on)); // R_TRIG
fb_stop_Fi(
    Execute := rtrig_stop_Fi.Q,
    Deceleration := gc_r_Stop_dec_Fi,
    Axis := v_FeedIndexer,
    Active => b_stop_act_Fi); // MC_Stop
b_start_goto_Fi R= fb_stop_Fi.Done;
b_stop_Fi_done := fb_stop_Fi.Done;

// NETWORK 5
//   b_stop_Az: the command of stop the motion
//   b_remote_on: in the remote mode
//   b_local_on: in the local mode
//   b_scc_maintain: the command of stowing the antenna at 20_degrees
//   b_scc_stow: the command of stowing the antenna at 90_degrees
rtrig_stop_goto_az(CLK := b_stop_Az AND (b_remote_on OR b_local_on)); // R_TRIG
b_scc_maintain R= rtrig_stop_goto_az.Q;
b_start_goto_az R= rtrig_stop_goto_az.Q;
b_scc_stow R= rtrig_stop_goto_az.Q;

// NETWORK 6
//   b_remote_on: in the remote mode
//   b_local_on: in the local mode
//   b_scc_maintain: the command of stowing the antenna at 20_degrees
//   b_scc_stow: the command of stowing the antenna at 90_degrees
rtrig_stop_goto_el(CLK := b_stop_El AND (b_remote_on OR b_local_on)); // R_TRIG
b_scc_maintain R= rtrig_stop_goto_el.Q;
b_start_goto_el R= rtrig_stop_goto_el.Q;
b_scc_stow R= rtrig_stop_goto_el.Q;

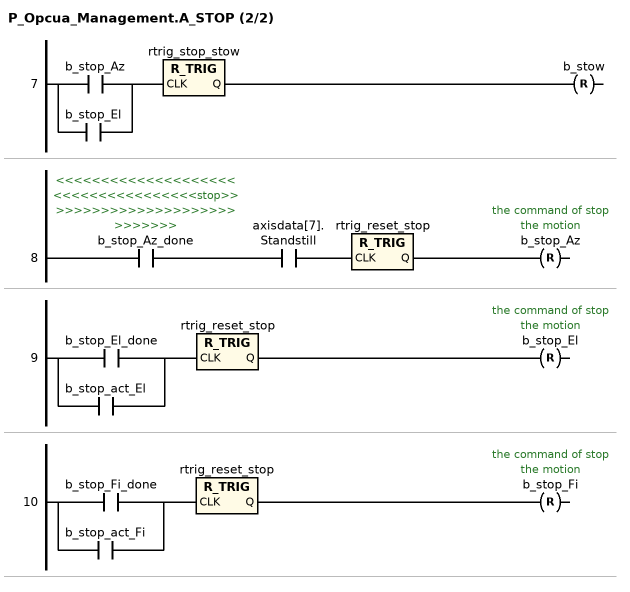
// NETWORK 7
rtrig_stop_stow(CLK := b_stop_Az OR b_stop_El); // R_TRIG
b_stow R= rtrig_stop_stow.Q;

// NETWORK 8
//   b_stop_Az_done: <<<<<<<<<<<<<<<<<<<<<<<<<<<<<<<<<<<<stop>>>>>>>>>>>>>>>>>>>>>>>>>>>>>
//   b_stop_Az: the command of stop the motion
rtrig_reset_stop(CLK := b_stop_Az_done AND axisdata[7].Standstill); // R_TRIG
b_stop_Az R= rtrig_reset_stop.Q;

// NETWORK 9
//   b_stop_El: the command of stop the motion
rtrig_reset_stop(CLK := b_stop_El_done OR b_stop_act_El); // R_TRIG
b_stop_El R= rtrig_reset_stop.Q;

// NETWORK 10
//   b_stop_Fi: the command of stop the motion
rtrig_reset_stop(CLK := b_stop_Fi_done OR b_stop_act_Fi); // R_TRIG
b_stop_Fi R= rtrig_reset_stop.Q;
END_ACTION

END_PROGRAM

// IndraMotionMlc1/Application/POUs/Panel Function/DANCE_OFF
PROGRAM DANCE_OFF
VAR
	R_TRIG_0: R_TRIG;
	dance_enable: BOOL;
	R_TRIG_1: R_TRIG;
	MC_Power_0: MC_Power;
	MC_MoveAbsolute_0: MC_MoveAbsolute;
	R_TRIG_2: R_TRIG;
	MC_MoveAbsolute_1: MC_MoveAbsolute;
	R_TRIG_3: R_TRIG;
	MC_MoveAbsolute_2: MC_MoveAbsolute;
	R_TRIG_4: R_TRIG;
	dance_step1: BOOL;
	MC_MoveAbsolute_3: MC_MoveAbsolute;
	R_TRIG_5: R_TRIG;
	dance_step2: BOOL;
	MC_MoveAbsolute_4: MC_MoveAbsolute;
	R_TRIG_6: R_TRIG;
	TON_0: TON;
	R_TRIG_7: R_TRIG;
	TON_1: TON;
	dance_step3: BOOL;
	TON_2: TON;
	dance_step4: BOOL;
	MC_MoveAbsolute_5: MC_MoveAbsolute;
	R_TRIG_8: R_TRIG;
	TON_3: TON;
	dance_step5: BOOL;
	MC_MoveAbsolute_6: MC_MoveAbsolute;
	R_TRIG_9: R_TRIG;
	TON_4: TON;
	dance_step6: BOOL;
	MC_MoveAbsolute_7: MC_MoveAbsolute;
	R_TRIG_10: R_TRIG;
	TON_5: TON;
	dance_step7: BOOL;
	R_TRIG_11: R_TRIG;
	dance_step8: BOOL;
	MC_MoveAbsolute_8: MC_MoveAbsolute;
	R_TRIG_12: R_TRIG;
	TON_6: TON;
	F_TRIG_0: F_TRIG;
	TON_7: TON;
	R_TRIG_13: R_TRIG;
	dance_step9: BOOL;
	R_TRIG_14: R_TRIG;
	TON_8: TON;
	TON_9: TON;
	R_TRIG_15: R_TRIG;
	TON_10: TON;
	dance_step10: BOOL;
	TON_11: TON;
END_VAR

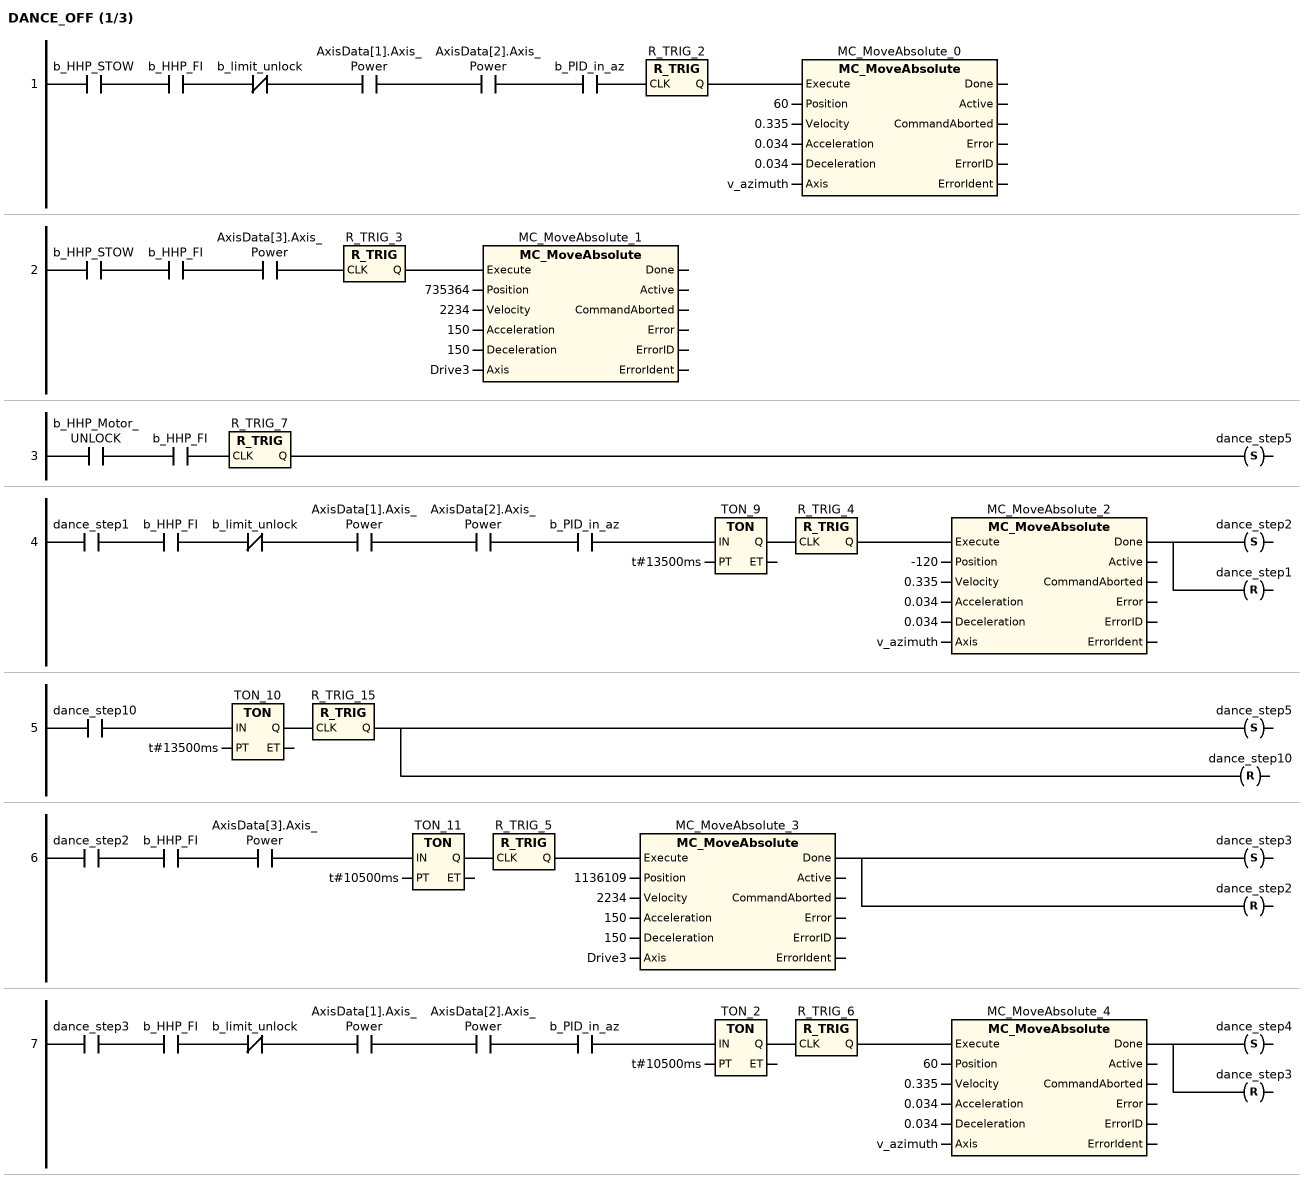
// NETWORK 1
R_TRIG_2(CLK := b_HHP_STOW AND b_HHP_FI AND NOT b_limit_unlock AND AxisData[1].Axis_Power AND AxisData[2].Axis_Power AND b_PID_in_az); // R_TRIG
MC_MoveAbsolute_0(
    Execute := R_TRIG_2.Q,
    Position := 60,
    Velocity := 0.335,
    Acceleration := 0.034,
    Deceleration := 0.034,
    Axis := v_azimuth); // MC_MoveAbsolute

// NETWORK 2
R_TRIG_3(CLK := b_HHP_STOW AND b_HHP_FI AND AxisData[3].Axis_Power); // R_TRIG
MC_MoveAbsolute_1(
    Execute := R_TRIG_3.Q,
    Position := 735364,
    Velocity := 2234,
    Acceleration := 150,
    Deceleration := 150,
    Axis := Drive3); // MC_MoveAbsolute

// NETWORK 3
R_TRIG_7(CLK := b_HHP_Motor_UNLOCK AND b_HHP_FI); // R_TRIG
dance_step5 S= R_TRIG_7.Q;

// NETWORK 4
TON_9(IN := dance_step1 AND b_HHP_FI AND NOT b_limit_unlock AND AxisData[1].Axis_Power AND AxisData[2].Axis_Power AND b_PID_in_az, PT := t#13500ms); // TON
R_TRIG_4(CLK := TON_9.Q); // R_TRIG
MC_MoveAbsolute_2(
    Execute := R_TRIG_4.Q,
    Position := -120,
    Velocity := 0.335,
    Acceleration := 0.034,
    Deceleration := 0.034,
    Axis := v_azimuth); // MC_MoveAbsolute
dance_step2 S= MC_MoveAbsolute_2.Done;
dance_step1 R= MC_MoveAbsolute_2.Done;

// NETWORK 5
TON_10(IN := dance_step10, PT := t#13500ms); // TON
R_TRIG_15(CLK := TON_10.Q); // R_TRIG
dance_step5 S= R_TRIG_15.Q;
dance_step10 R= R_TRIG_15.Q;

// NETWORK 6
TON_11(IN := dance_step2 AND b_HHP_FI AND AxisData[3].Axis_Power, PT := t#10500ms); // TON
R_TRIG_5(CLK := TON_11.Q); // R_TRIG
MC_MoveAbsolute_3(
    Execute := R_TRIG_5.Q,
    Position := 1136109,
    Velocity := 2234,
    Acceleration := 150,
    Deceleration := 150,
    Axis := Drive3); // MC_MoveAbsolute
dance_step3 S= MC_MoveAbsolute_3.Done;
dance_step2 R= MC_MoveAbsolute_3.Done;

// NETWORK 7
TON_2(IN := dance_step3 AND b_HHP_FI AND NOT b_limit_unlock AND AxisData[1].Axis_Power AND AxisData[2].Axis_Power AND b_PID_in_az, PT := t#10500ms); // TON
R_TRIG_6(CLK := TON_2.Q); // R_TRIG
MC_MoveAbsolute_4(
    Execute := R_TRIG_6.Q,
    Position := 60,
    Velocity := 0.335,
    Acceleration := 0.034,
    Deceleration := 0.034,
    Axis := v_azimuth); // MC_MoveAbsolute
dance_step4 S= MC_MoveAbsolute_4.Done;
dance_step3 R= MC_MoveAbsolute_4.Done;

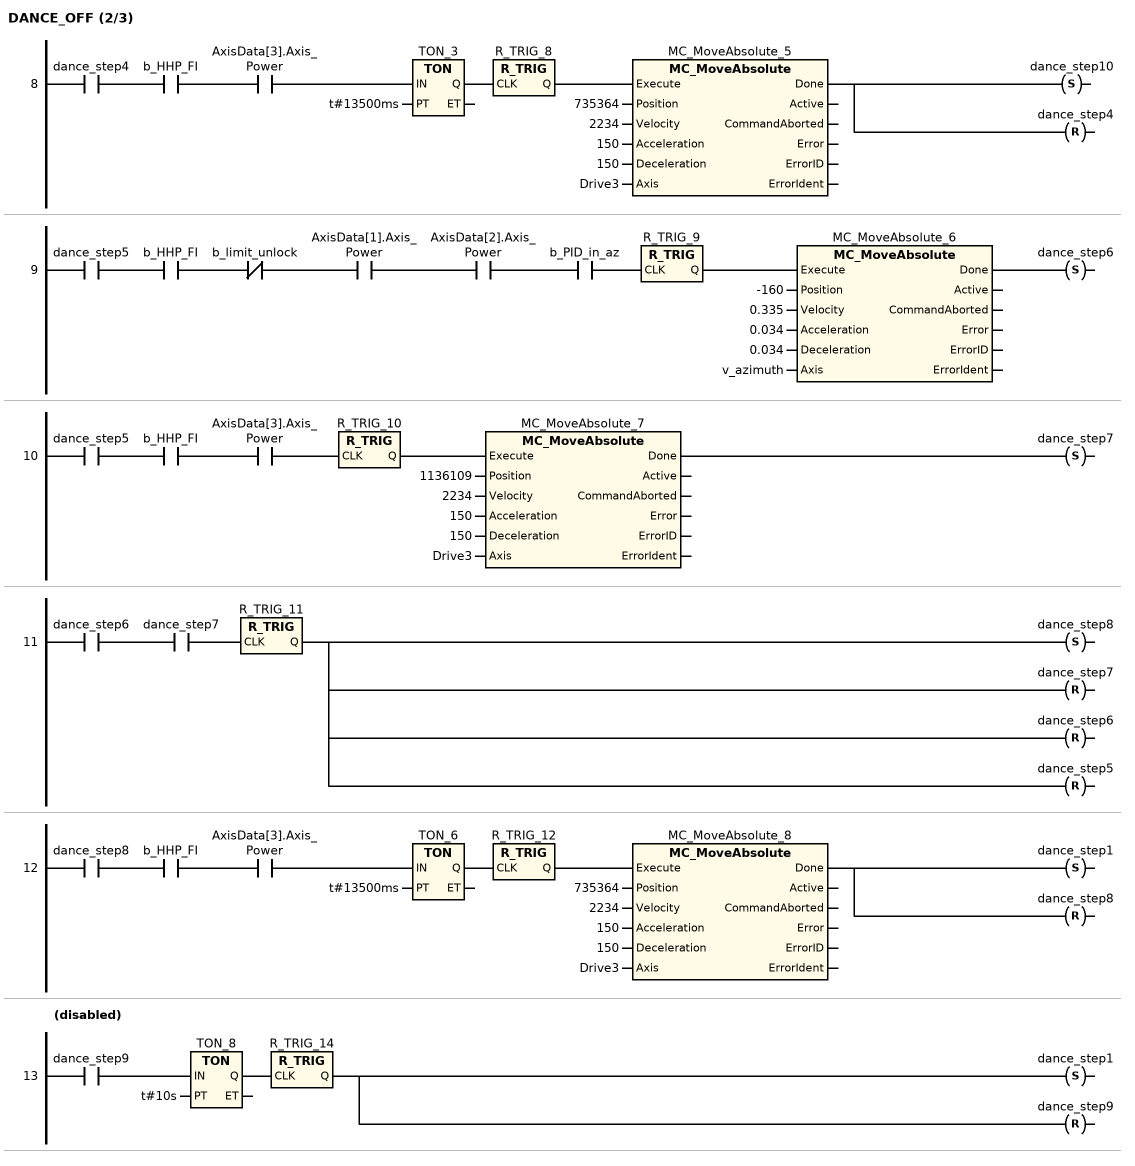
// NETWORK 8
TON_3(IN := dance_step4 AND b_HHP_FI AND AxisData[3].Axis_Power, PT := t#13500ms); // TON
R_TRIG_8(CLK := TON_3.Q); // R_TRIG
MC_MoveAbsolute_5(
    Execute := R_TRIG_8.Q,
    Position := 735364,
    Velocity := 2234,
    Acceleration := 150,
    Deceleration := 150,
    Axis := Drive3); // MC_MoveAbsolute
dance_step10 S= MC_MoveAbsolute_5.Done;
dance_step4 R= MC_MoveAbsolute_5.Done;

// NETWORK 9
R_TRIG_9(CLK := dance_step5 AND b_HHP_FI AND NOT b_limit_unlock AND AxisData[1].Axis_Power AND AxisData[2].Axis_Power AND b_PID_in_az); // R_TRIG
MC_MoveAbsolute_6(
    Execute := R_TRIG_9.Q,
    Position := -160,
    Velocity := 0.335,
    Acceleration := 0.034,
    Deceleration := 0.034,
    Axis := v_azimuth); // MC_MoveAbsolute
dance_step6 S= MC_MoveAbsolute_6.Done;

// NETWORK 10
R_TRIG_10(CLK := dance_step5 AND b_HHP_FI AND AxisData[3].Axis_Power); // R_TRIG
MC_MoveAbsolute_7(
    Execute := R_TRIG_10.Q,
    Position := 1136109,
    Velocity := 2234,
    Acceleration := 150,
    Deceleration := 150,
    Axis := Drive3); // MC_MoveAbsolute
dance_step7 S= MC_MoveAbsolute_7.Done;

// NETWORK 11
R_TRIG_11(CLK := dance_step6 AND dance_step7); // R_TRIG
dance_step8 S= R_TRIG_11.Q;
dance_step7 R= R_TRIG_11.Q;
dance_step6 R= R_TRIG_11.Q;
dance_step5 R= R_TRIG_11.Q;

// NETWORK 12
TON_6(IN := dance_step8 AND b_HHP_FI AND AxisData[3].Axis_Power, PT := t#13500ms); // TON
R_TRIG_12(CLK := TON_6.Q); // R_TRIG
MC_MoveAbsolute_8(
    Execute := R_TRIG_12.Q,
    Position := 735364,
    Velocity := 2234,
    Acceleration := 150,
    Deceleration := 150,
    Axis := Drive3); // MC_MoveAbsolute
dance_step1 S= MC_MoveAbsolute_8.Done;
dance_step8 R= MC_MoveAbsolute_8.Done;

// NETWORK 13 (disabled)
// TON_8(IN := dance_step9, PT := t#10s); // TON
// R_TRIG_14(CLK := TON_8.Q); // R_TRIG
// dance_step1 S= R_TRIG_14.Q;
// dance_step9 R= R_TRIG_14.Q;

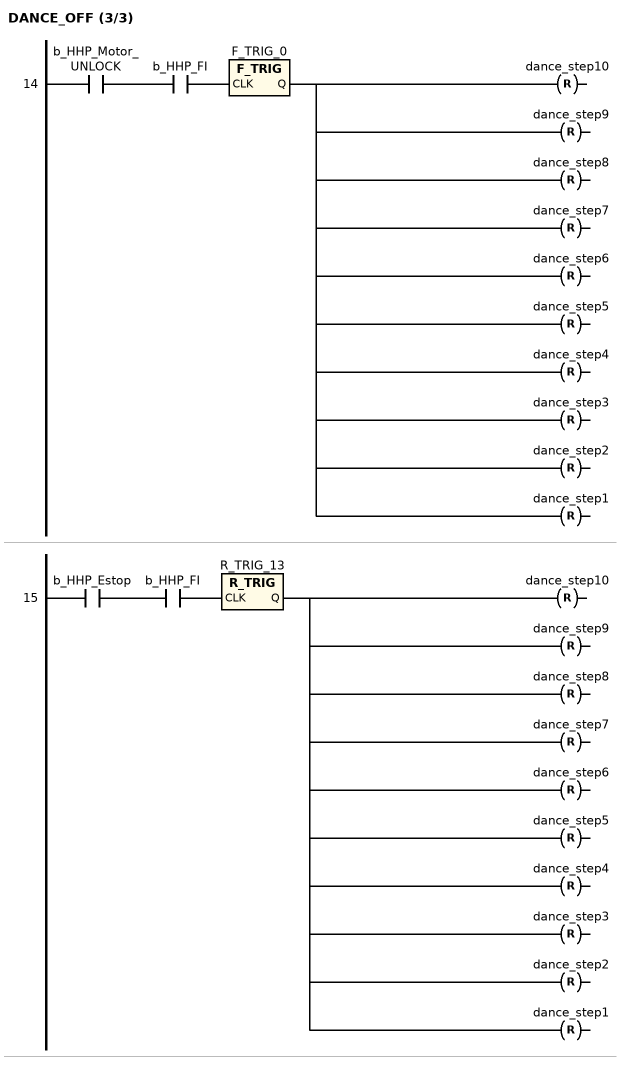
// NETWORK 14
F_TRIG_0(CLK := b_HHP_Motor_UNLOCK AND b_HHP_FI); // F_TRIG
dance_step10 R= F_TRIG_0.Q;
dance_step9 R= F_TRIG_0.Q;
dance_step8 R= F_TRIG_0.Q;
dance_step7 R= F_TRIG_0.Q;
dance_step6 R= F_TRIG_0.Q;
dance_step5 R= F_TRIG_0.Q;
dance_step4 R= F_TRIG_0.Q;
dance_step3 R= F_TRIG_0.Q;
dance_step2 R= F_TRIG_0.Q;
dance_step1 R= F_TRIG_0.Q;

// NETWORK 15
R_TRIG_13(CLK := b_HHP_Estop AND b_HHP_FI); // R_TRIG
dance_step10 R= R_TRIG_13.Q;
dance_step9 R= R_TRIG_13.Q;
dance_step8 R= R_TRIG_13.Q;
dance_step7 R= R_TRIG_13.Q;
dance_step6 R= R_TRIG_13.Q;
dance_step5 R= R_TRIG_13.Q;
dance_step4 R= R_TRIG_13.Q;
dance_step3 R= R_TRIG_13.Q;
dance_step2 R= R_TRIG_13.Q;
dance_step1 R= R_TRIG_13.Q;

END_PROGRAM

// IndraMotionMlc1/Application/POUs/Panel Function/FI_TEST
PROGRAM FI_TEST
VAR
	MC_Power_0: MC_Power;
	fi_enable1: BOOL;
	MC_Power_1: MC_Power;
	fi_enable2: BOOL;
	MC_TorqueControl_0: MC_TorqueControl;
	fi_torque1: BOOL;
	MC_TorqueControl_1: MC_TorqueControl;
	fi_torque2: BOOL;
	MC_MoveVelocity_0: MC_MoveVelocity;
	fi_move1: BOOL;
	fi_vel1: REAL;
	BLINK_0: BLINK;
	BLINK_1: BLINK;
	MC_MoveVelocity_1: MC_MoveVelocity;
	fi_move2: BOOL;
	fi_vel2: REAL;
	BLINK_2: BLINK;
	MB_ReadRealParameter_0: MB_ReadRealParameter;
	fi_encoder1: REAL;
	MB_ReadRealParameter_1: MB_ReadRealParameter;
	fi_encoder2: REAL;
	MC_Stop_0: MC_Stop;
	MC_Stop_1: MC_Stop;
	fi_stop: BOOL;
	R_TRIG_0: R_TRIG;
	R_TRIG_1: R_TRIG;
	R_TRIG_2: R_TRIG;
	R_TRIG_3: R_TRIG;
	MB_ReadParameter_0: MB_ReadParameter;
	MB_ReadParameter_1: MB_ReadParameter;
	fi_brake1: DWORD;
	fi_brake2: DWORD;
END_VAR

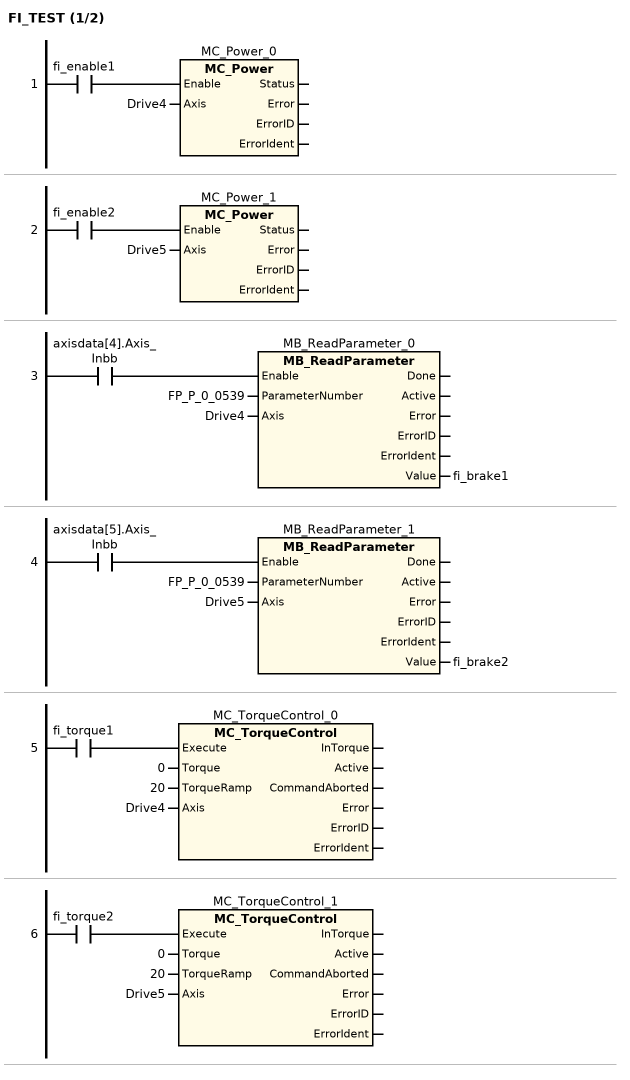
// NETWORK 1
MC_Power_0(Enable := fi_enable1, Axis := Drive4); // MC_Power

// NETWORK 2
MC_Power_1(Enable := fi_enable2, Axis := Drive5); // MC_Power

// NETWORK 3
MB_ReadParameter_0(
    Enable := axisdata[4].Axis_Inbb,
    ParameterNumber := FP_P_0_0539,
    Axis := Drive4,
    Value => fi_brake1); // MB_ReadParameter

// NETWORK 4
MB_ReadParameter_1(
    Enable := axisdata[5].Axis_Inbb,
    ParameterNumber := FP_P_0_0539,
    Axis := Drive5,
    Value => fi_brake2); // MB_ReadParameter

// NETWORK 5
MC_TorqueControl_0(Execute := fi_torque1, Torque := 0, TorqueRamp := 20, Axis := Drive4); // MC_TorqueControl

// NETWORK 6
MC_TorqueControl_1(Execute := fi_torque2, Torque := 0, TorqueRamp := 20, Axis := Drive5); // MC_TorqueControl

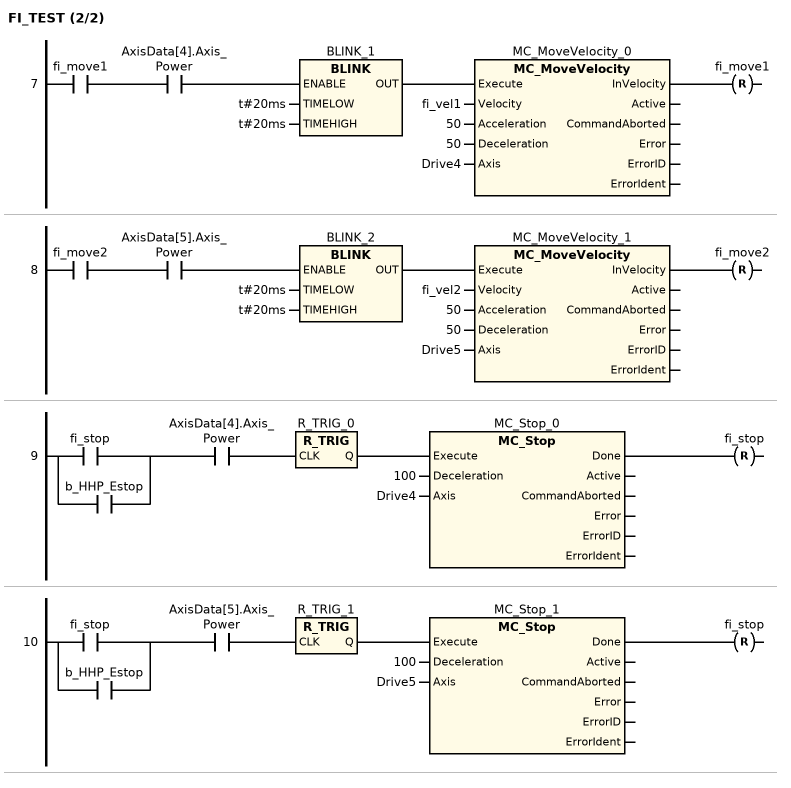
// NETWORK 7
BLINK_1(ENABLE := fi_move1 AND AxisData[4].Axis_Power, TIMELOW := t#20ms, TIMEHIGH := t#20ms); // BLINK
MC_MoveVelocity_0(
    Execute := BLINK_1.OUT,
    Velocity := fi_vel1,
    Acceleration := 50,
    Deceleration := 50,
    Axis := Drive4); // MC_MoveVelocity
fi_move1 R= MC_MoveVelocity_0.InVelocity;

// NETWORK 8
BLINK_2(ENABLE := fi_move2 AND AxisData[5].Axis_Power, TIMELOW := t#20ms, TIMEHIGH := t#20ms); // BLINK
MC_MoveVelocity_1(
    Execute := BLINK_2.OUT,
    Velocity := fi_vel2,
    Acceleration := 50,
    Deceleration := 50,
    Axis := Drive5); // MC_MoveVelocity
fi_move2 R= MC_MoveVelocity_1.InVelocity;

// NETWORK 9
R_TRIG_0(CLK := (fi_stop OR b_HHP_Estop) AND AxisData[4].Axis_Power); // R_TRIG
MC_Stop_0(Execute := R_TRIG_0.Q, Deceleration := 100, Axis := Drive4); // MC_Stop
fi_stop R= MC_Stop_0.Done;

// NETWORK 10
R_TRIG_1(CLK := (fi_stop OR b_HHP_Estop) AND AxisData[5].Axis_Power); // R_TRIG
MC_Stop_1(Execute := R_TRIG_1.Q, Deceleration := 100, Axis := Drive5); // MC_Stop
fi_stop R= MC_Stop_1.Done;

END_PROGRAM

// IndraMotionMlc1/Application/POUs/Panel Function/P_LED
(*
This progrom is bulit for lighting the led in the panelbox which describe the limit.
1)If the angle is reach the limit value,we use the Function Block MB_WriteParameter to setting 
special value to the parameter FP_P_0_0304 of the relative drive.so that the led will be lighted.
2)Besides,when the position of azimuth axis is at the zone,60 degrees nearby the limit,the led of azimuth will flicker every 2 seconds.
Similar with azimuth,the elevation LED will flicker at the 5-degrees-zone nearby limit,and the FeedIndexer LED will flicker at the 30-degrees-zone nearby limit.
*)
PROGRAM P_LED
VAR
(*the definition of Blink function blocks*)
	fb_blink_LED_az: BLINK;
	fb_blink_write_az: BLINK;
	fb_blink_LED_el: BLINK;
	fb_blink_write_el: BLINK;
	fb_blink_LED_FI: BLINK;
	fb_blink_write_FI: BLINK;
	t_LED_az: TIME;
	t_LED_el: TIME;
	t_LED_FI: TIME;
	b_LED_az: BOOL;
	b_LED_el: BOOL;
	b_LED_FI: BOOL;
(*the definition of function blocks for Writing p304 Parameter*)
	fb_write_p304_d2: MB_WriteParameter;(*the I/O of azimuth LED is on drive2*)
	fb_write_p304_d4: MB_WriteParameter;(*the I/O of elevation LED is on drive4*)
	fb_write_p304_d5: MB_WriteParameter;(*the I/O of FeedIndexer LED is on drive5*)
(*when the P304 parameter equal to 512,only the 9th on the I/O is set;
when the P304 parameter equal to 1024,only the 10th on the I/O is set;
when the P304 parameter equal to 0,all the I/O is reset;*)
	i_p304_az: INT;
	i_p304_el: INT;
	i_p304_FI: INT;
END_VAR




IF b_local_on=TRUE THEN
	b_local_led:=TRUE;
ELSE
	b_local_led:=FALSE;
END_IF

IF b_remote_on=TRUE THEN
	b_remote_led:=TRUE;
ELSE
	b_remote_led:=FALSE;
END_IF

IF b_ESTOP_door=TRUE THEN
	b_estop_led :=TRUE;
ELSE
	b_estop_led :=FALSE;
END_IF

   IF master_status.4 =FALSE THEN
	   b_normal_led:=TRUE;
	   b_error_led:=FALSE;
   ELSE
   	   b_normal_led:=FALSE;
	   b_error_led:=TRUE;
   END_IF


(*
IF b_local_on=TRUE THEN
(*<<<<<<<<<<<<<<<<<<<<<<<<<<<<<<<<LED Of azimuth>>>>>>>>>>>>>>>>>>>>>>>>>>>>>>>>>*)
	IF r_pos_az>=0 AND r_pos_az<=180 THEN
		i_p304_az:=0;
	ELSIF r_pos_az>180 AND r_pos_az<358.5 THEN
		t_LED_az:=T#2.2s;
		IF b_LED_az= TRUE THEN
			i_p304_az:=0;
		ELSE
			i_p304_az:=512;
		END_IF
	ELSIF r_pos_az>=358.5 THEN
		i_p304_az:=512;
	ELSIF r_pos_az<0 AND r_pos_az>-178.5 THEN
		t_LED_az:=T#2.2s;
		IF b_LED_az= TRUE THEN
			i_p304_az:=0;
		ELSE
			i_p304_az:=1024;
		END_IF
	ELSIF r_pos_az<=-178.5 THEN
		i_p304_az:=1024;
	END_IF
(*<<<<<<<<<<<<<<<<<<<<<<<<<<<<<<<<LED Of elevation>>>>>>>>>>>>>>>>>>>>>>>>>>>>>>>>>*)
	IF r_pos_el>=25 AND r_pos_el<=80 THEN
		i_p304_el:=0;
	ELSIF r_pos_el>80 AND r_pos_el<=90.1 THEN
		t_LED_el:=T#2.2s;
		IF b_LED_el= TRUE THEN
			i_p304_el:=0;
		ELSE
			i_p304_el:=512;
		END_IF
	ELSIF r_pos_el>90.1 THEN
		i_p304_el:=512;
	ELSIF r_pos_el>25 AND r_pos_el<=15 THEN
		t_LED_el:=T#2.2s;
		IF b_LED_el= TRUE THEN
			i_p304_el:=0;
		ELSE
			i_p304_el:=1024;
		END_IF
	ELSIF r_pos_el<15 THEN
		i_p304_el:=1024;
	END_IF
(*<<<<<<<<<<<<<<<<<<<<<<<<<<<<<<<<LED Of FeedIndexer>>>>>>>>>>>>>>>>>>>>>>>>>>>>>>>>>*)
	IF r_pos_FI>=-120 AND r_pos_FI<=120 THEN
		i_p304_FI:=0;
	ELSIF r_pos_FI>120 AND r_pos_FI<=178.5 THEN
		t_LED_FI:=T#2.2s;
		IF b_LED_FI= TRUE THEN
			i_p304_FI:=0;
		ELSE
			i_p304_FI:=512;
		END_IF
	ELSIF r_pos_FI>178.5 THEN
		i_p304_FI:=512;
	ELSIF r_pos_FI<-120 AND r_pos_FI>=-178.5 THEN
		t_LED_FI:=T#2.2s;
		IF b_LED_FI= TRUE THEN
			i_p304_FI:=0;
		ELSE
			i_p304_FI:=1024;
		END_IF
	ELSIF r_pos_FI<-178.5 THEN
		i_p304_FI:=1024;
	END_IF
ELSE
(*if not at local situation,the LED is dark*)
(*For testing LED,write i_p304_az:=1536;i_p304_el:=1536;i_p304_FI:=1536;*)
	i_p304_az:=0;
	i_p304_el:=0;
	i_p304_FI:=0;
END_IF

(*transfer the sub-program A_w_P304 to white value to the parameter FP_P_0_0304*)
P_LED.A_w_P304;*)

ACTION A_w_P304:
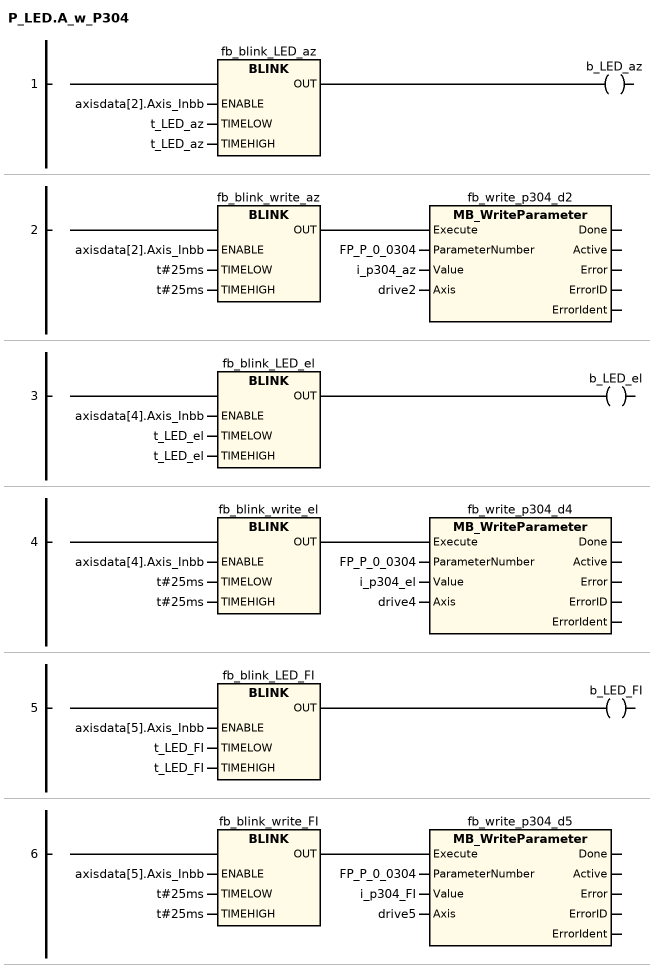
// NETWORK 1
fb_blink_LED_az(ENABLE := axisdata[2].Axis_Inbb, TIMELOW := t_LED_az, TIMEHIGH := t_LED_az); // BLINK
b_LED_az := fb_blink_LED_az.OUT;

// NETWORK 2
fb_blink_write_az(ENABLE := axisdata[2].Axis_Inbb, TIMELOW := t#25ms, TIMEHIGH := t#25ms); // BLINK
fb_write_p304_d2(
    Execute := fb_blink_write_az.OUT,
    ParameterNumber := FP_P_0_0304,
    Value := i_p304_az,
    Axis := drive2); // MB_WriteParameter

// NETWORK 3
fb_blink_LED_el(ENABLE := axisdata[4].Axis_Inbb, TIMELOW := t_LED_el, TIMEHIGH := t_LED_el); // BLINK
b_LED_el := fb_blink_LED_el.OUT;

// NETWORK 4
fb_blink_write_el(ENABLE := axisdata[4].Axis_Inbb, TIMELOW := t#25ms, TIMEHIGH := t#25ms); // BLINK
fb_write_p304_d4(
    Execute := fb_blink_write_el.OUT,
    ParameterNumber := FP_P_0_0304,
    Value := i_p304_el,
    Axis := drive4); // MB_WriteParameter

// NETWORK 5
fb_blink_LED_FI(ENABLE := axisdata[5].Axis_Inbb, TIMELOW := t_LED_FI, TIMEHIGH := t_LED_FI); // BLINK
b_LED_FI := fb_blink_LED_FI.OUT;

// NETWORK 6
fb_blink_write_FI(ENABLE := axisdata[5].Axis_Inbb, TIMELOW := t#25ms, TIMEHIGH := t#25ms); // BLINK
fb_write_p304_d5(
    Execute := fb_blink_write_FI.OUT,
    ParameterNumber := FP_P_0_0304,
    Value := i_p304_FI,
    Axis := drive5); // MB_WriteParameter
END_ACTION

END_PROGRAM

// IndraMotionMlc1/Application/POUs/Panel Function/P_Lock_Panel_TCP
(*This program is bulit for lock the antenna for stow and maintain,and for unlock the antenna.
It mainly contains goto function,the control of AC moter,and the protect for safety*)
PROGRAM P_Lock_Panel_TCP
VAR

(*<<<<<<<<<<<<<<<<<<<the allow for the lock moter>>>>>>>>>>>>>>>>>*)
	b_lock_allow_0: BOOL;
	b_lock_allow_20: BOOL;
(*the definition of rise trigger,The function block R_TRIG detects a rising edge. *)
	rtrig_lock_stow: R_TRIG;
	rtrig_lock_maintain: R_TRIG;
	rtrig_reset_TCP_unlock: R_TRIG;
	rtrig_reset_TCP_lock: R_TRIG;
	rtrig_enable_unlock: R_TRIG;
(*The function block Timer On Delay implements a turn-on delay*)
	ton_stow_0: TON;
	ton_maintain_20: TON;
	ton_reset_lock: TON;
	ton_reset_unlock: TON;
(*the fixed position according to the hole*)
	r_postion_stow: REAL;
	r_position_maintain: REAL;
(*move the elevation to the fixed position*)
	fb_move_AZ_0: MC_MoveAbsolute;
	fb_move_el_20: MC_MoveAbsolute;
	fb_self_reset_stow: R_TRIG;
	fb_ton_self_reset_stow: TON;
	b_lock_allow_21: BOOL;
	fb_self_reset_maintain: R_TRIG;
	fb_ton_self_reset_maintain: TON;
	b_off_stow: R_TRIG;
	b_off_maintain: R_TRIG;
	fb_move_EL_0: MC_MoveAbsolute;
END_VAR

(*<<<<<<<<<<<<<<<<<<<<write the stow and maintain position according to IP>>>>>>>>>>>>>>>>>>>>>>>>>>>>>>>>>>>>*)
(*every antenna maybe has the different stow position and maintain position from the others*)
str_1xx:=RIGHT(str_MLC_ip,3);(*for get the last 3 number of IP in MLC*)
IF str_1xx='101' THEN
	r_postion_stow:=0;
	r_position_maintain:=20.15;
ELSIF str_1xx='102' THEN
	r_postion_stow:=0;
	r_position_maintain:=20.820;
ELSIF str_1xx='103' THEN
	r_postion_stow:=0;
	r_position_maintain:=20.950;
ELSIF str_1xx='104' THEN
	r_postion_stow:=0;
	r_position_maintain:=20.9;
ELSIF str_1xx='105' THEN
	r_postion_stow:=0;
	r_position_maintain:=20.930;
ELSIF str_1xx='106' THEN
	r_postion_stow:=0;
	r_position_maintain:=20.800;
ELSIF str_1xx='107' THEN
	r_postion_stow:=90.00;
	r_position_maintain:=20.850;
ELSIF str_1xx='108' THEN
	r_postion_stow:=90.00;
	r_position_maintain:=21.100;
ELSIF str_1xx='109' THEN
	r_postion_stow:=90.00;
	r_position_maintain:=21.000;
ELSIF str_1xx='110' THEN
	r_postion_stow:=0;
	r_position_maintain:=21.000;
ELSIF str_1xx='111' THEN
	r_postion_stow:=0;
	r_position_maintain:=21.000;
ELSIF str_1xx='112' THEN
	r_postion_stow:=0;
	r_position_maintain:=21.100;
ELSIF str_1xx='113' THEN
	r_postion_stow:=0;
	r_position_maintain:=21.000;
ELSIF str_1xx='114' THEN
	r_postion_stow:=0;
	r_position_maintain:=21.000;
ELSIF str_1xx='115' THEN
	r_postion_stow:=0;
	r_position_maintain:=21.000;
ELSIF str_1xx='116' THEN
	r_postion_stow:=0;
	r_position_maintain:=21.000;
ELSIF str_1xx='117' THEN
	r_postion_stow:=0;
	r_position_maintain:=21.000;
ELSIF str_1xx='118' THEN
	r_postion_stow:=0;
	r_position_maintain:=20.950;
ELSIF str_1xx='119' THEN
	r_postion_stow:=0;
	r_position_maintain:=20.950;
ELSIF str_1xx='120' THEN
	r_postion_stow:=0;
	r_position_maintain:=21.000;
ELSIF str_1xx='121' THEN
	r_postion_stow:=0;
	r_position_maintain:=21.000;
ELSIF str_1xx='122' THEN
	r_postion_stow:=0;
	r_position_maintain:=21.000;
ELSIF str_1xx='123' THEN
	r_postion_stow:=0;
	r_position_maintain:=21.000;
ELSIF str_1xx='124' THEN
	r_postion_stow:=0;
	r_position_maintain:=21.000;
ELSIF str_1xx='125' THEN
	r_postion_stow:=0;
	r_position_maintain:=21.000;
ELSIF str_1xx='126' THEN
	r_postion_stow:=0;
	r_position_maintain:=21.000;
ELSIF str_1xx='127' THEN
	r_postion_stow:=0;
	r_position_maintain:=21.000;
ELSIF str_1xx='128' THEN
	r_postion_stow:=0;
	r_position_maintain:=21.000;
ELSIF str_1xx='129' THEN
	r_postion_stow:=0;
	r_position_maintain:=21.000;
ELSIF str_1xx='130' THEN
	r_postion_stow:=0;
	r_position_maintain:=20.950;
ELSIF str_1xx='131' THEN
	r_postion_stow:=0;
	r_position_maintain:=21.000;
ELSIF str_1xx='132' THEN
	r_postion_stow:=0;
	r_position_maintain:=21.000;
ELSIF str_1xx='133' THEN
	r_postion_stow:=0;
	r_position_maintain:=21.000;
ELSIF str_1xx='134' THEN
	r_postion_stow:=0;
	r_position_maintain:=21.000;
ELSIF str_1xx='135' THEN
	r_postion_stow:=0.00;
	r_position_maintain:=21.000;
ELSIF str_1xx='136' THEN
	r_postion_stow:=0.00;
	r_position_maintain:=21.000;

(*test*)
ELSIF str_1xx='1.1' THEN
	r_postion_stow:=0.00;
	r_position_maintain:=20.9;
ELSE
	r_postion_stow:=0;
	r_position_maintain:=11;
END_IF
(*<<<<<<<<<<<<<<<<<<<<<<<<<<<<<<<<if the elevation position is nearby the fixed value,then allow the lock action>>>>>>>>>>>>>>>>>>>>>>>>>>>>>>>>>>>>>>>>>>>>>>>>>>>*)
IF ABS(axisdata[1].rActualPosition_i-0)<0.01 THEN
	b_lock_allow_0:=TRUE;
ELSE
	b_lock_allow_0:=FALSE;
END_IF

IF b_stow_pin_limit_lock = FALSE AND ABS(axisdata[1].rActualPosition_i-r_postion_stow)< 0.1 THEN
	b_stow_lock:=TRUE;
ELSE
	b_stow_lock:=FALSE;
END_IF;

P_Lock_Panel_TCP.A_LOCK();

ACTION A_LOCK:
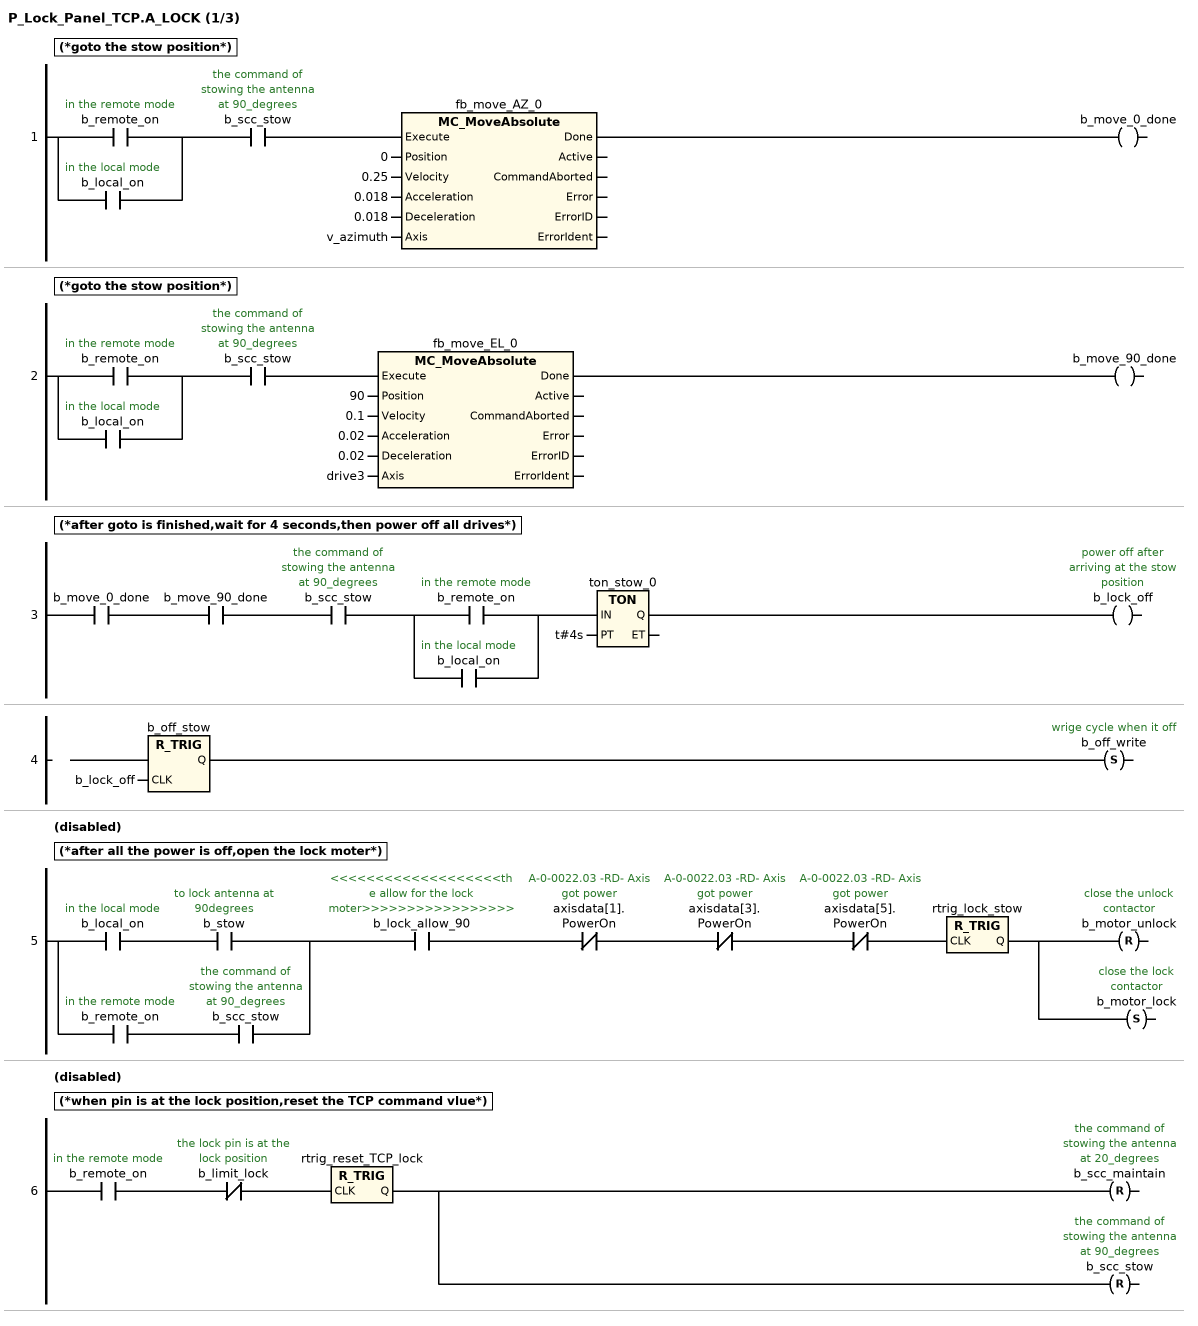
// NETWORK 1
//   fb_move_AZ_0: move the elevation to the fixed position
//   b_remote_on: in the remote mode
//   b_local_on: in the local mode
//   b_scc_stow: the command of stowing the antenna at 90_degrees
//   v_azimuth: Virtual axis "v_elevation" with axis number 8
// label: (*goto the stow position*)
fb_move_AZ_0(
    Execute := (b_remote_on OR b_local_on) AND b_scc_stow,
    Position := 0,
    Velocity := 0.25,
    Acceleration := 0.018,
    Deceleration := 0.018,
    Axis := v_azimuth); // MC_MoveAbsolute
b_move_0_done := fb_move_AZ_0.Done;

// NETWORK 2
//   fb_move_EL_0: move the elevation to the fixed position
//   b_remote_on: in the remote mode
//   b_local_on: in the local mode
//   b_scc_stow: the command of stowing the antenna at 90_degrees
//   drive3: Virtual axis "v_elevation" with axis number 8
// label: (*goto the stow position*)
fb_move_EL_0(
    Execute := (b_remote_on OR b_local_on) AND b_scc_stow,
    Position := 90,
    Velocity := 0.1,
    Acceleration := 0.02,
    Deceleration := 0.02,
    Axis := drive3); // MC_MoveAbsolute
b_move_90_done := fb_move_EL_0.Done;

// NETWORK 3
//   ton_stow_0: The function block Timer On Delay implements a turn-on delay
//   b_scc_stow: the command of stowing the antenna at 90_degrees
//   b_remote_on: in the remote mode
//   b_local_on: in the local mode
//   b_lock_off: power off after arriving at the stow position
// label: (*after goto is finished,wait for 4 seconds,then power off all drives*)
ton_stow_0(IN := b_move_0_done AND b_move_90_done AND b_scc_stow AND (b_remote_on OR b_local_on), PT := t#4s); // TON
b_lock_off := ton_stow_0.Q;

// NETWORK 4
//   b_lock_off: power off after arriving at the stow position
//   b_off_write: wrige cycle when it off
b_off_stow(CLK := b_lock_off); // R_TRIG
b_off_write S= b_off_stow.Q;

// NETWORK 5 (disabled)
//   rtrig_lock_stow: the definition of rise trigger,The function block R_TRIG detects a rising edge.
//   b_local_on: in the local mode
//   b_stow: to lock antenna at 90degrees
//   b_remote_on: in the remote mode
//   b_scc_stow: the command of stowing the antenna at 90_degrees
//   b_lock_allow_90: <<<<<<<<<<<<<<<<<<<the allow for the lock moter>>>>>>>>>>>>>>>>>
//   axisdata[1].PowerOn: A-0-0022.03 -RD- Axis got power
//   axisdata[3].PowerOn: A-0-0022.03 -RD- Axis got power
//   axisdata[5].PowerOn: A-0-0022.03 -RD- Axis got power
//   b_motor_unlock: close the unlock contactor
//   b_motor_lock: close the lock contactor
// label: (*after all the power is off,open the lock moter*)
// rtrig_lock_stow(CLK := (b_local_on AND b_stow OR b_remote_on AND b_scc_stow) AND b_lock_allow_90 AND NOT axisdata[1].PowerOn AND NOT axisdata[3].PowerOn AND NOT axisdata[5].PowerOn); // R_TRIG
// b_motor_unlock R= rtrig_lock_stow.Q;
// b_motor_lock S= rtrig_lock_stow.Q;

// NETWORK 6 (disabled)
//   b_remote_on: in the remote mode
//   b_limit_lock: the lock pin is at the lock position
//   b_scc_maintain: the command of stowing the antenna at 20_degrees
//   b_scc_stow: the command of stowing the antenna at 90_degrees
// label: (*when pin is at the lock position,reset the TCP command vlue*)
// rtrig_reset_TCP_lock(CLK := b_remote_on AND NOT b_limit_lock); // R_TRIG
// b_scc_maintain R= rtrig_reset_TCP_lock.Q;
// b_scc_stow R= rtrig_reset_TCP_lock.Q;

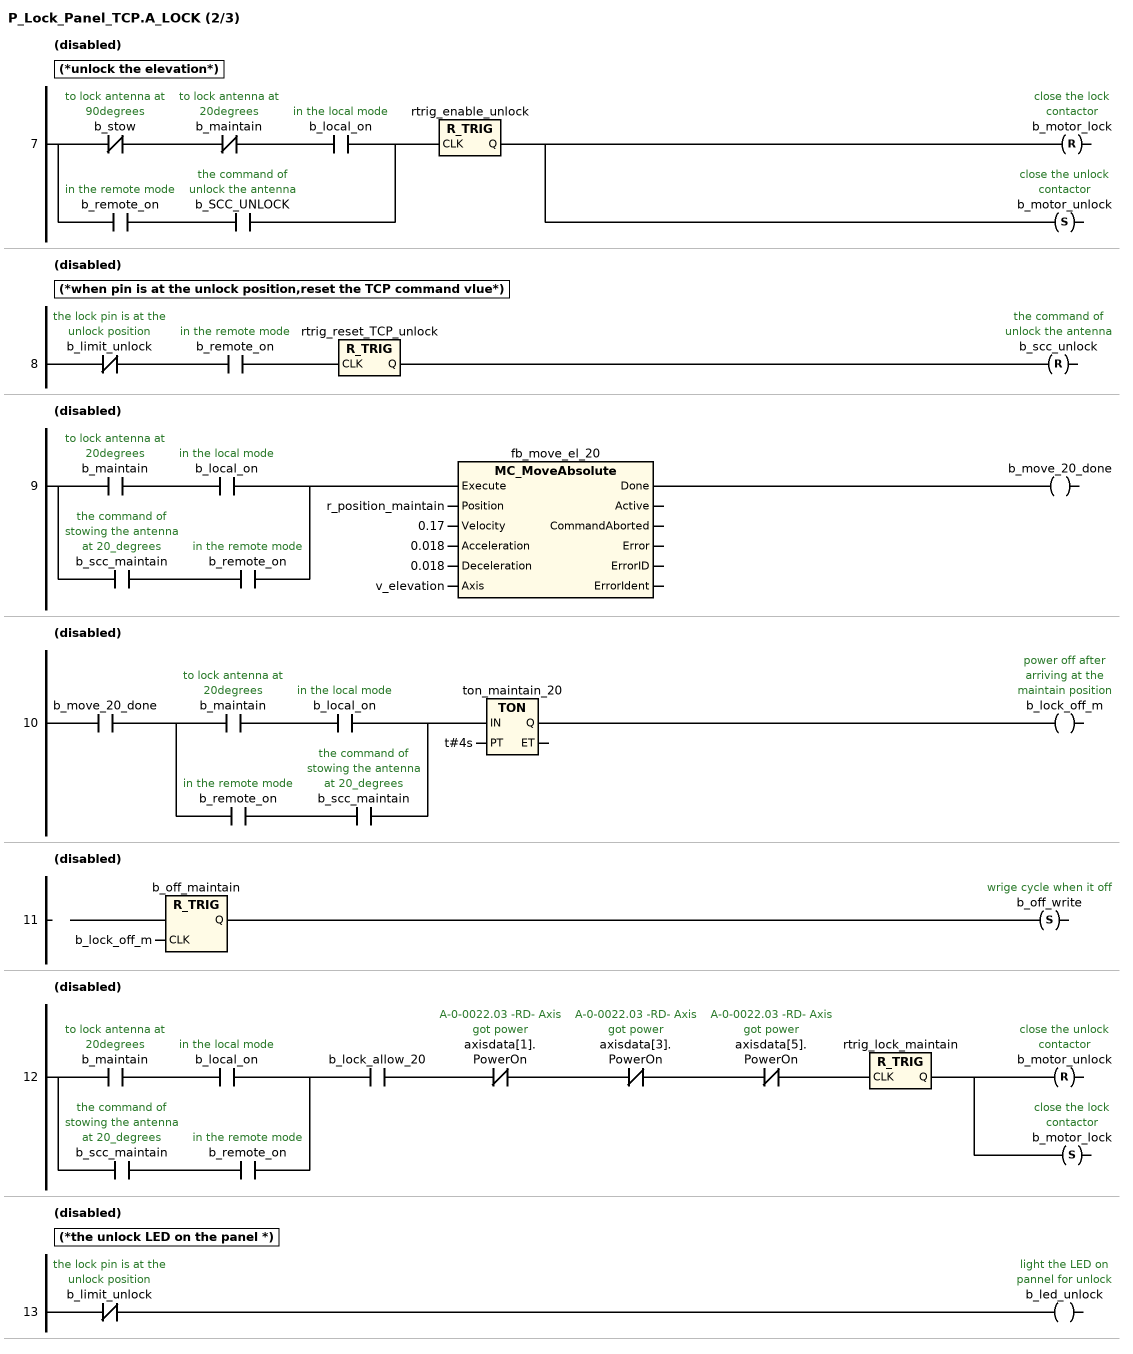
// NETWORK 7 (disabled)
//   b_stow: to lock antenna at 90degrees
//   b_maintain: to lock antenna at 20degrees
//   b_local_on: in the local mode
//   b_remote_on: in the remote mode
//   b_SCC_UNLOCK: the command of unlock the antenna
//   b_motor_lock: close the lock contactor
//   b_motor_unlock: close the unlock contactor
// label: (*unlock the elevation*)
// rtrig_enable_unlock(CLK := NOT b_stow AND NOT b_maintain AND b_local_on OR b_remote_on AND b_SCC_UNLOCK); // R_TRIG
// b_motor_lock R= rtrig_enable_unlock.Q;
// b_motor_unlock S= rtrig_enable_unlock.Q;

// NETWORK 8 (disabled)
//   b_limit_unlock: the lock pin is at the unlock position
//   b_remote_on: in the remote mode
//   b_scc_unlock: the command of unlock the antenna
// label: (*when pin is at the unlock position,reset the TCP command vlue*)
// rtrig_reset_TCP_unlock(CLK := NOT b_limit_unlock AND b_remote_on); // R_TRIG
// b_scc_unlock R= rtrig_reset_TCP_unlock.Q;

// NETWORK 9 (disabled)
//   b_maintain: to lock antenna at 20degrees
//   b_local_on: in the local mode
//   b_scc_maintain: the command of stowing the antenna at 20_degrees
//   b_remote_on: in the remote mode
//   v_elevation: Virtual axis "v_elevation" with axis number 8
// fb_move_el_20(
//     Execute := b_maintain AND b_local_on OR b_scc_maintain AND b_remote_on,
//     Position := r_position_maintain,
//     Velocity := 0.17,
//     Acceleration := 0.018,
//     Deceleration := 0.018,
//     Axis := v_elevation); // MC_MoveAbsolute
// b_move_20_done := fb_move_el_20.Done;

// NETWORK 10 (disabled)
//   b_maintain: to lock antenna at 20degrees
//   b_local_on: in the local mode
//   b_remote_on: in the remote mode
//   b_scc_maintain: the command of stowing the antenna at 20_degrees
//   b_lock_off_m: power off after arriving at the maintain position
// ton_maintain_20(IN := b_move_20_done AND (b_maintain AND b_local_on OR b_remote_on AND b_scc_maintain), PT := t#4s); // TON
// b_lock_off_m := ton_maintain_20.Q;

// NETWORK 11 (disabled)
//   b_lock_off_m: power off after arriving at the maintain position
//   b_off_write: wrige cycle when it off
// b_off_maintain(CLK := b_lock_off_m); // R_TRIG
// b_off_write S= b_off_maintain.Q;

// NETWORK 12 (disabled)
//   b_maintain: to lock antenna at 20degrees
//   b_local_on: in the local mode
//   b_scc_maintain: the command of stowing the antenna at 20_degrees
//   b_remote_on: in the remote mode
//   axisdata[1].PowerOn: A-0-0022.03 -RD- Axis got power
//   axisdata[3].PowerOn: A-0-0022.03 -RD- Axis got power
//   axisdata[5].PowerOn: A-0-0022.03 -RD- Axis got power
//   b_motor_unlock: close the unlock contactor
//   b_motor_lock: close the lock contactor
// rtrig_lock_maintain(CLK := (b_maintain AND b_local_on OR b_scc_maintain AND b_remote_on) AND b_lock_allow_20 AND NOT axisdata[1].PowerOn AND NOT axisdata[3].PowerOn AND NOT axisdata[5].PowerOn); // R_TRIG
// b_motor_unlock R= rtrig_lock_maintain.Q;
// b_motor_lock S= rtrig_lock_maintain.Q;

// NETWORK 13 (disabled)
//   b_limit_unlock: the lock pin is at the unlock position
//   b_led_unlock: light the LED on pannel for unlock
// label: (*the unlock LED on the panel *)
// b_led_unlock := NOT b_limit_unlock;

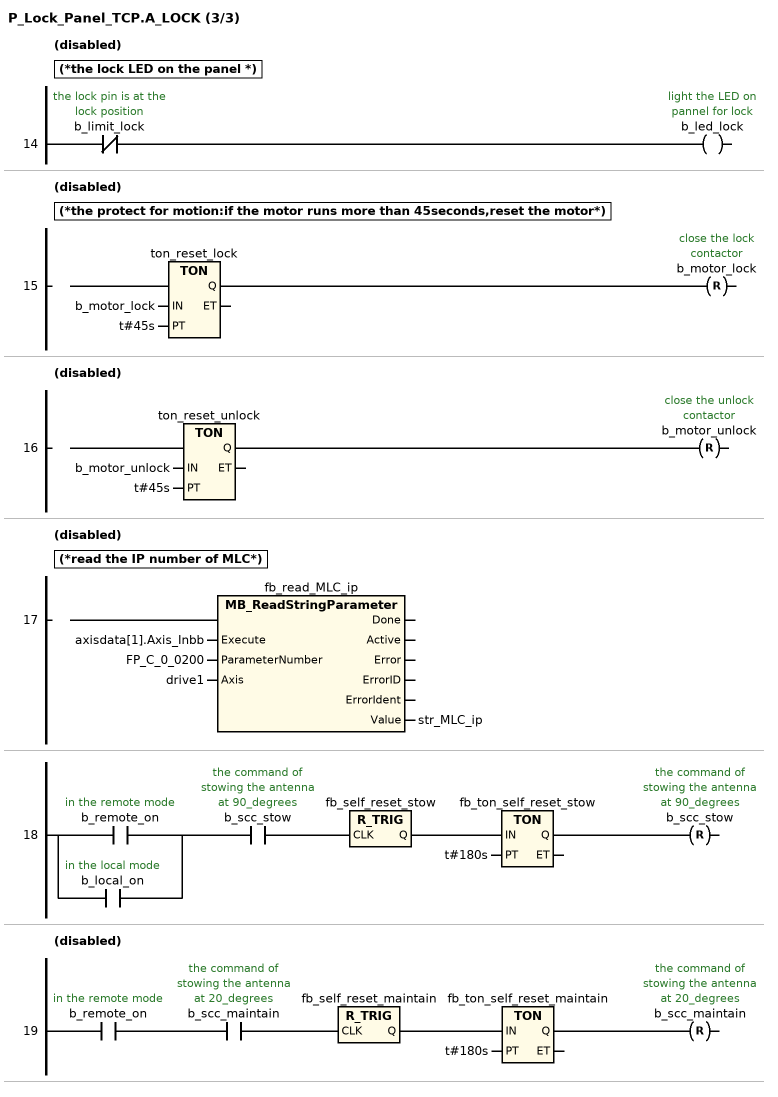
// NETWORK 14 (disabled)
//   b_limit_lock: the lock pin is at the lock position
//   b_led_lock: light the LED on pannel for lock
// label: (*the lock LED on the panel *)
// b_led_lock := NOT b_limit_lock;

// NETWORK 15 (disabled)
//   b_motor_lock: close the lock contactor
// label: (*the protect for motion:if the motor runs more than 45seconds,reset the motor*)
// ton_reset_lock(IN := b_motor_lock, PT := t#45s); // TON
// b_motor_lock R= ton_reset_lock.Q;

// NETWORK 16 (disabled)
//   b_motor_unlock: close the unlock contactor
// ton_reset_unlock(IN := b_motor_unlock, PT := t#45s); // TON
// b_motor_unlock R= ton_reset_unlock.Q;

// NETWORK 17 (disabled)
//   axisdata[1].Axis_Inbb: A-0-0021.13 -RD- Axis is ready for power to the amplifier (bb)
//   FP_C_0_0200: Engineering, IP address
//   drive1: Real axis "Drive1" with axis number 1
//   str_MLC_ip: IP number in MLC
// label: (*read the IP number of MLC*)
// fb_read_MLC_ip(
//     Execute := axisdata[1].Axis_Inbb,
//     ParameterNumber := FP_C_0_0200,
//     Axis := drive1,
//     Value => str_MLC_ip); // MB_ReadStringParameter

// NETWORK 18
//   b_remote_on: in the remote mode
//   b_local_on: in the local mode
//   b_scc_stow: the command of stowing the antenna at 90_degrees
fb_self_reset_stow(CLK := (b_remote_on OR b_local_on) AND b_scc_stow); // R_TRIG
fb_ton_self_reset_stow(IN := fb_self_reset_stow.Q, PT := t#180s); // TON
b_scc_stow R= fb_ton_self_reset_stow.Q;

// NETWORK 19 (disabled)
//   b_remote_on: in the remote mode
//   b_scc_maintain: the command of stowing the antenna at 20_degrees
// fb_self_reset_maintain(CLK := b_remote_on AND b_scc_maintain); // R_TRIG
// fb_ton_self_reset_maintain(IN := fb_self_reset_maintain.Q, PT := t#180s); // TON
// b_scc_maintain R= fb_ton_self_reset_maintain.Q;
END_ACTION

END_PROGRAM

// IndraMotionMlc1/Application/POUs/Panel Function/P_Panel_Jog
PROGRAM P_Panel_Jog
VAR
(*<<<<<<<<<<<<<<<azimuth>>>>>>>>>>>>>>>>*)
	r_vel_az: REAL;
	fb_panel_vel_az: MC_MoveVelocity;
	fb_panel_stop_az: MC_Stop;
	rtrig_panel_stop_az: R_TRIG;
	fb_blink_az: BLINK;
(*<<<<<<<<<<<<<<<elevation>>>>>>>>>>>>>>>*)
	r_vel_el: REAL;
	fb_panel_vel_el: MC_MoveVelocity;
	fb_panel_stop_el: MC_Stop;
	rtrig_panel_stop_el: R_TRIG;
	fb_blink_el: BLINK;
(*<<<<<<<<<<<<<FeedIndexer>>>>>>>>>>>>>>>>>*)
	r_vel_FI: REAL;
	fb_panel_vel_FI: MC_MoveVelocity;
	fb_panel_stop_FI: MC_Stop;
	rtrig_panel_stop_FI: R_TRIG;
	fb_blink_FI: BLINK;
(*the moving fuction into P_panel_jog program for FAT test and SAT test *)
	fb_test_move_az: MC_MoveAbsolute;
	fb_test_move_el: MC_MoveAbsolute;
	fb_test_move_FI: MC_MoveAbsolute;
	b_test_az: BOOL;
	b_test_el: BOOL;
	b_test_FI: BOOL;
	r_test_az: REAL;
	r_test_el: REAL;
	r_test_FI: REAL;
	r_test_vel_az:REAL;
	r_test_vel_el:REAL;
	r_test_vel_FI:REAL;
	b_test_az_r: BOOL;
	r_test_az_r: REAL;
	fb_test_relative_az: MC_MoveRelative;
	fb_test_relative_FI: MC_MoveRelative;
	r_test_FI_r: REAL;
	b_test_FI_r: BOOL;
END_VAR



(*<<<<<<<<<<<<<<<<<<<<<<<<<add the limit of the panel control>>>>>>>>>>>>>>>>>>>>>>>>*)
IF r_pos_az >= 358.5 THEN
	b_clockwise_AZ:= FALSE;
END_IF
IF r_pos_az <= -178.5 THEN
	b_cclockwise_AZ:= FALSE;
END_IF
IF r_pos_el >=90.1 THEN
	b_up_el:= FALSE;
END_IF
IF r_pos_el <=15 THEN
	b_down_el:=FALSE;
END_IF
IF r_pos_FI >= 178.5 THEN
	b_clockwise_FI:= FALSE;
END_IF
IF r_pos_FI <= -178.5 THEN
	b_cclockwise_FI:= FALSE;
END_IF

(*<<<<<<<<<<<<<<<<<<<<<<<set the azimuth speed value>>>>>>>>>>>>>>>>>>>>>>>>>>*)
IF b_clockwise_AZ = TRUE THEN
	IF b_speed_az = TRUE THEN
		r_vel_az:=0.5;
	ELSE
		r_vel_az:=0.17;
	END_IF
	IF r_pos_az>355 THEN
		r_vel_az:=0.17;
	END_IF
END_IF
IF b_cclockwise_AZ = TRUE THEN
	IF b_speed_az = TRUE THEN
		r_vel_az:=-0.5;
	ELSE
		r_vel_az:=-0.17;
	END_IF
	IF r_pos_az<-175 THEN
		r_vel_az:=-0.17;
	END_IF
END_IF
(*<<<<<<<<<<<<<<<<<<<<<<<set the elevation speed value>>>>>>>>>>>>>>>>>>>>>>>>>>*)
IF b_up_el =TRUE THEN
	IF b_speed_el = TRUE THEN
		r_vel_el:=0.17;
	ELSE
		r_vel_el:=0.05;
	END_IF
	IF r_pos_el>89 THEN
		r_vel_el:=0.05;
	END_IF
END_IF
IF b_down_el =TRUE THEN
	IF b_speed_el = TRUE THEN
		r_vel_el:=-0.17;
	ELSE
		r_vel_el:=-0.05;
	END_IF
	IF r_pos_el<16 THEN
		r_vel_el:=-0.05;
	END_IF
END_IF
(*<<<<<<<<<<<<<<<<<<<<<<<set the FeedIndexer speed value>>>>>>>>>>>>>>>>>>>>>>>>>>*)
IF b_clockwise_FI = TRUE THEN
	IF b_speed_FI = TRUE THEN
		r_vel_FI:=0.5;
	ELSE
		r_vel_FI:=0.17;
	END_IF
	IF r_pos_FI>175 THEN
		r_vel_FI:=0.17;
	END_IF
END_IF
IF b_cclockwise_FI = TRUE THEN
	IF b_speed_FI = TRUE THEN
		r_vel_FI:=-0.5;
	ELSE
		r_vel_FI:=-0.17;
	END_IF
	IF r_pos_FI<-175 THEN
		r_vel_FI:=-0.17;
	END_IF
END_IF

P_Panel_Jog.A_axes_running;

